KUKA KRL program: ps_b_ltb_res_c02.src, ps_b_ltb_res_c02.dat

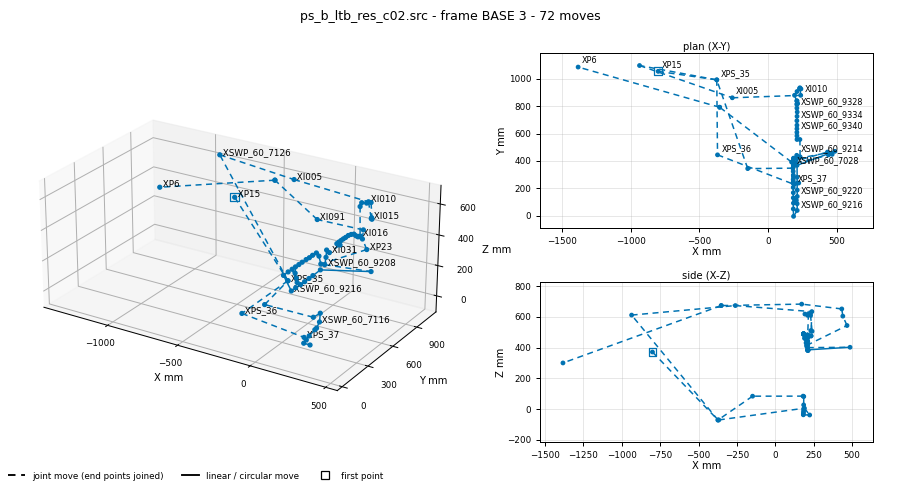
[picture p0: tool path of ps_b_ltb_res_c02.src in frame BASE 3, 72 of 73 moves have a stored position in this frame; points joined in program order, loops and branches not executed]
--- ps_b_ltb_res_c02.src ---
&ACCESS RVO1
&COMMENT Solda Axor LTB
DEF ps_b_ltb_res_c02( )

  ;FOLD INI;%{PE}%V2.2.2,%MKUKATPBASIS,%CINIT,%VCOMMON,%P
  ;FOLD BAS INI;%{PE}%V2.2.2,%MKUKATPBASIS,%CINIT,%VINIT,%P
  INTERRUPT DECL 3 WHEN $STOPMESS==TRUE DO IR_STOPM ( )
  INTERRUPT ON 3
  BAS (#INITMOV,0 )
  ;ENDFOLD
  ;FOLD A20 INI;%{E}%V2.2.2,%MKUKATPA20,%CINIT,%VINIT,%P
  IF ARC20==TRUE THEN
    A20 (ARC_INI)
    INTERRUPT DECL 6 WHEN $CYCFLAG[3]==FALSE DO A20(TECH_STOP2)
  ENDIF
  ;ENDFOLD
  ;FOLD A10 INI;%{E}%V2.2.2,%MKUKATPARC,%CINIT,%VINIT,%P
  IF A10_OPTION==#ACTIVE THEN
    INTERRUPT DECL 4 WHEN $CYCFLAG[2]==FALSE DO A10 (#APPL_ERROR)
    INTERRUPT DECL 7 WHEN A_ARC_SWI==#ACTIVE DO A10 (#ARC_SEAM)
    INTERRUPT DECL 5 WHEN A_FLY_ARC==TRUE DO A10 (#HPU_ARC)
    INTERRUPT  ON 5
    A10_INI ( )
  ENDIF
  ;ENDFOLD
  ;FOLD GRIPPER INI;%{E}%V2.2.2,%MKUKATPGRIPPER,%CINIT,%VINIT,%P
  USER_GRP(0,DUMMY,DUMMY,GDEFAULT)
  ;ENDFOLD
  ;FOLD SPOT INI;%{E}%V.2.2,%MKUKATPSPOT,%CINIT,%VINIT,%P
  USERSPOT(#INIT)
  ;ENDFOLD
  ;FOLD TOUCHSENSE INI;%{E}%V2.2.2,%MKUKATPTS,%CINIT,%VINIT,%P
  IF H70_OPTION THEN
    INTERRUPT DECL 15 WHEN $MEAS_PULSE[TOUCH_I[TOUCH_ACTIVE].IN_NR] DO H70 (6,CD0 )
    INTERRUPT DECL 16 WHEN $ZERO_MOVE DO H70 (7,CD0 )
    INTERRUPT DECL 17 WHEN $TECHPAR_C[FG_TOUCH,8]>0.5 DO H70 (8,CD0)
    H70 (1,CD0 )
  ENDIF
  ;ENDFOLD
  ;FOLD USER INI;%{P}%V2.2.2,%MKUKATPUSER,%CINIT,%VINIT,%P
  ;Make your modifications here
  ;ENDFOLD
  ;ENDFOLD

; Caracterizacao dos meios de producao
; Changes: Solda Respot - ATEGO - STB
; Versao Atual: 26/03/2016
; Ferramenta : Gun C02
; Name: P13.060-R4

chk_w3_wechs_ok ( )    ; CHECK GUN C02

IF(NOT(GHOST())) THEN
IF MaxStandMenge(3) THEN
  MaxStandmengeErreicht()
ENDIF

IF Elektrodenwechsel(3) THEN
e_Fraes3()
ENDIF
ENDIF

;FOLD OUT 868 'Perfil Livre Estacao'  State= FALSE ;%{PE}%R 4.1.16,%MKUKATPBASIS,%COUT,%VOUTX,%P 2:868, 3:'Perfil Livre Estacao', 5:FALSE, 6:
$OUT[868]=FALSE
;ENDFOLD

;FOLD PTP P15  Vel= 100 % PDAT2 Tool[1]:GUN C1 Base[3]:Atego/Axor;%{PE}%R 4.1.16,%MKUKATPBASIS,%CMOVE,%VPTP,%P 1:PTP, 2:P15, 3:, 5:100, 7:PDAT2
$BWDSTART = FALSE
PDAT_ACT=PPDAT2
BAS(#PTP_DAT)
FDAT_ACT=FP15
BAS(#FRAMES)
BAS(#VEL_PTP,100)
PTP XP15
;ENDFOLD

;FOLD ; Liga Intertravamento 1 c/ R01;%{PE}%R 4.1.16,%MKUKATPBASIS,%CCOMMENT,%VNORMAL,%P 2:Liga Intertravamento 1 c/ R01
;ENDFOLD
;FOLD ; Liga Intertravamento 10 c/ R02;%{PE}%R 4.1.16,%MKUKATPBASIS,%CCOMMENT,%VNORMAL,%P 2:Liga Intertravamento 10 c/ R02
;ENDFOLD
;FOLD Kollision.Ueberwachung_1_Ein ;%{PE}%MKUKATPUSER
COLLSTOP( 1, 1 ) ;INTERRUPTUEBERWACHT
;ENDFOLD
;FOLD Kollision.Monitoring_AREA_4_On ;%{PE}%MKUKATPUSER
COLLSTOP( 10, 1 ) ;NICHT INTERRUPTUEBERWACHT
;ENDFOLD


;FOLD ; Liga Intertravamento 3 c/ R03;%{PE}%R 4.1.16,%MKUKATPBASIS,%CCOMMENT,%VNORMAL,%P 2:Liga Intertravamento 7 c/ R03
;ENDFOLD
;FOLD Kollision.Ueberwachung_3_Ein ;%{PE}%MKUKATPUSER
COLLSTOP( 3, 1 ) ;INTERRUPTUEBERWACHT
;ENDFOLD


;FOLD PTP PS_35 CONT Vel= 100 % PDAT29 Tool[3]:GUN C02 Base[3]:Atego/Axor;%{PE}%R 4.1.16,%MKUKATPBASIS,%CMOVE,%VPTP,%P 1:PTP, 2:PS_35, 3:C_PTP, 5:100, 7:PDAT29
$BWDSTART = FALSE
PDAT_ACT=PPDAT29
BAS(#PTP_DAT)
FDAT_ACT=FPS_35
BAS(#FRAMES)
BAS(#VEL_PTP,100)
PTP XPS_35 C_PTP
;ENDFOLD
;FOLD PTP PS_36 CONT Vel= 100 % PDAT30 Tool[3]:GUN C02 Base[3]:Atego/Axor;%{PE}%R 4.1.16,%MKUKATPBASIS,%CMOVE,%VPTP,%P 1:PTP, 2:PS_36, 3:C_PTP, 5:100, 7:PDAT30
$BWDSTART = FALSE
PDAT_ACT=PPDAT30
BAS(#PTP_DAT)
FDAT_ACT=FPS_36
BAS(#FRAMES)
BAS(#VEL_PTP,100)
PTP XPS_36 C_PTP
;ENDFOLD
;FOLD PTP PS_37 CONT Vel= 100 % PDAT31 Tool[3]:GUN C02 Base[3]:Atego/Axor;%{PE}%R 4.1.16,%MKUKATPBASIS,%CMOVE,%VPTP,%P 1:PTP, 2:PS_37, 3:C_PTP, 5:100, 7:PDAT31
$BWDSTART = FALSE
PDAT_ACT=PPDAT31
BAS(#PTP_DAT)
FDAT_ACT=FPS_37
BAS(#FRAMES)
BAS(#VEL_PTP,100)
PTP XPS_37 C_PTP
;ENDFOLD
;FOLD PTP PS_38 CONT Vel= 100 % PDAT32 Tool[3]:GUN C02 Base[3]:Atego/Axor;%{PE}%R 4.1.16,%MKUKATPBASIS,%CMOVE,%VPTP,%P 1:PTP, 2:PS_38, 3:C_PTP, 5:100, 7:PDAT32
$BWDSTART = FALSE
PDAT_ACT=PPDAT32
BAS(#PTP_DAT)
FDAT_ACT=FPS_38
BAS(#FRAMES)
BAS(#VEL_PTP,100)
PTP XPS_38 C_PTP
;ENDFOLD


;FOLD LIN SWP_60_7106 CPDAT22 SPOT Gun= 3 RETR CLS PgNo1= 197 ACTIVE= 1 Tool[3]:GUN C02 Base[3]:Atego/Axor;%{PE}%R 4.1.12,%MKUKATPSPOT,%CSPOT,%VLIN,%P 1:LIN, 2:SWP_60_7106, 3:, 5:2, 7:CPDAT22, 10:3, 12:#FIRST, 14:#CLO, 16:197, 18:1, 20:0, 22:0, 24:1, 25:NORMAL
$BWDSTART = FALSE
LDAT_ACT=LCPDAT22
BAS(#CP_DAT)
FDAT_ACT=FSWP_60_7106
BAS(#FRAMES)
BAS(#VEL_CP,LCPDAT22.VEL)
S_ACT.GUN=3
S_ACT.PAIR=SDEFAULT.PAIR
S_ACT.RETR=#CLO
S_ACT.CLO_TM=1
S_ACT.PGNO1=197
S_ACT.PGNO2=SDEFAULT.PGNO2
S_ACT.PRESS1=SDEFAULT.PRESS1
S_ACT.PRESS2=SDEFAULT.PRESS2
S_READY=FALSE
LIN XSWP_60_7106
USERSPOT(#SPOT, S_ACT)
WAIT FOR S_READY
;ENDFOLD


;FOLD LIN SWP_60_7108 CPDAT23 SPOT Gun= 3 RETR CLS PgNo1= 197 ACTIVE= 1 Tool[3]:GUN C02 Base[3]:Atego/Axor;%{PE}%R 4.1.12,%MKUKATPSPOT,%CSPOT,%VLIN,%P 1:LIN, 2:SWP_60_7108, 3:, 5:2, 7:CPDAT23, 10:3, 12:#FIRST, 14:#CLO, 16:197, 18:1, 20:0, 22:0, 24:1, 25:NORMAL
$BWDSTART = FALSE
LDAT_ACT=LCPDAT23
BAS(#CP_DAT)
FDAT_ACT=FSWP_60_7108
BAS(#FRAMES)
BAS(#VEL_CP,LCPDAT23.VEL)
S_ACT.GUN=3
S_ACT.PAIR=SDEFAULT.PAIR
S_ACT.RETR=#CLO
S_ACT.CLO_TM=1
S_ACT.PGNO1=197
S_ACT.PGNO2=SDEFAULT.PGNO2
S_ACT.PRESS1=SDEFAULT.PRESS1
S_ACT.PRESS2=SDEFAULT.PRESS2
S_READY=FALSE
LIN XSWP_60_7108
USERSPOT(#SPOT, S_ACT)
WAIT FOR S_READY
;ENDFOLD

;FOLD LIN SWP_60_7110 CPDAT24 SPOT Gun= 3 RETR CLS PgNo1= 197 ACTIVE= 1 Tool[3]:GUN C02 Base[3]:Atego/Axor;%{PE}%R 4.1.12,%MKUKATPSPOT,%CSPOT,%VLIN,%P 1:LIN, 2:SWP_60_7110, 3:, 5:2, 7:CPDAT24, 10:3, 12:#FIRST, 14:#CLO, 16:197, 18:1, 20:0, 22:0, 24:1, 25:NORMAL
$BWDSTART = FALSE
LDAT_ACT=LCPDAT24
BAS(#CP_DAT)
FDAT_ACT=FSWP_60_7110
BAS(#FRAMES)
BAS(#VEL_CP,LCPDAT24.VEL)
S_ACT.GUN=3
S_ACT.PAIR=SDEFAULT.PAIR
S_ACT.RETR=#CLO
S_ACT.CLO_TM=1
S_ACT.PGNO1=197
S_ACT.PGNO2=SDEFAULT.PGNO2
S_ACT.PRESS1=SDEFAULT.PRESS1
S_ACT.PRESS2=SDEFAULT.PRESS2
S_READY=FALSE
LIN XSWP_60_7110
USERSPOT(#SPOT, S_ACT)
WAIT FOR S_READY
;ENDFOLD

;FOLD LIN SWP_60_7028 CPDAT25 SPOT Gun= 3 RETR CLS PgNo1= 197 ACTIVE= 1 Tool[3]:GUN C02 Base[3]:Atego/Axor;%{PE}%R 4.1.12,%MKUKATPSPOT,%CSPOT,%VLIN,%P 1:LIN, 2:SWP_60_7028, 3:, 5:2, 7:CPDAT25, 10:3, 12:#FIRST, 14:#CLO, 16:197, 18:1, 20:0, 22:0, 24:1, 25:NORMAL
$BWDSTART = FALSE
LDAT_ACT=LCPDAT25
BAS(#CP_DAT)
FDAT_ACT=FSWP_60_7028
BAS(#FRAMES)
BAS(#VEL_CP,LCPDAT25.VEL)
S_ACT.GUN=3
S_ACT.PAIR=SDEFAULT.PAIR
S_ACT.RETR=#CLO
S_ACT.CLO_TM=1
S_ACT.PGNO1=197
S_ACT.PGNO2=SDEFAULT.PGNO2
S_ACT.PRESS1=SDEFAULT.PRESS1
S_ACT.PRESS2=SDEFAULT.PRESS2
S_READY=FALSE
LIN XSWP_60_7028
USERSPOT(#SPOT, S_ACT)
WAIT FOR S_READY
;ENDFOLD

;FOLD LIN SWP_60_7114 CPDAT26 SPOT Gun= 3 RETR CLS PgNo1= 197 ACTIVE= 1 Tool[3]:GUN C02 Base[3]:Atego/Axor;%{PE}%R 4.1.12,%MKUKATPSPOT,%CSPOT,%VLIN,%P 1:LIN, 2:SWP_60_7114, 3:, 5:2, 7:CPDAT26, 10:3, 12:#FIRST, 14:#CLO, 16:197, 18:1, 20:0, 22:0, 24:1, 25:NORMAL
$BWDSTART = FALSE
LDAT_ACT=LCPDAT26
BAS(#CP_DAT)
FDAT_ACT=FSWP_60_7114
BAS(#FRAMES)
BAS(#VEL_CP,LCPDAT26.VEL)
S_ACT.GUN=3
S_ACT.PAIR=SDEFAULT.PAIR
S_ACT.RETR=#CLO
S_ACT.CLO_TM=1
S_ACT.PGNO1=197
S_ACT.PGNO2=SDEFAULT.PGNO2
S_ACT.PRESS1=SDEFAULT.PRESS1
S_ACT.PRESS2=SDEFAULT.PRESS2
S_READY=FALSE
LIN XSWP_60_7114
USERSPOT(#SPOT, S_ACT)
WAIT FOR S_READY
;ENDFOLD


;FOLD LIN SWP_60_7116 CPDAT27 SPOT Gun= 3 RETR CLS PgNo1= 197 ACTIVE= 1 Tool[3]:GUN C02 Base[3]:Atego/Axor;%{PE}%R 4.1.12,%MKUKATPSPOT,%CSPOT,%VLIN,%P 1:LIN, 2:SWP_60_7116, 3:, 5:2, 7:CPDAT27, 10:3, 12:#FIRST, 14:#CLO, 16:197, 18:1, 20:0, 22:0, 24:1, 25:NORMAL
$BWDSTART = FALSE
LDAT_ACT=LCPDAT27
BAS(#CP_DAT)
FDAT_ACT=FSWP_60_7116
BAS(#FRAMES)
BAS(#VEL_CP,LCPDAT27.VEL)
S_ACT.GUN=3
S_ACT.PAIR=SDEFAULT.PAIR
S_ACT.RETR=#CLO
S_ACT.CLO_TM=1
S_ACT.PGNO1=197
S_ACT.PGNO2=SDEFAULT.PGNO2
S_ACT.PRESS1=SDEFAULT.PRESS1
S_ACT.PRESS2=SDEFAULT.PRESS2
S_READY=FALSE
LIN XSWP_60_7116
USERSPOT(#SPOT, S_ACT)
WAIT FOR S_READY
;ENDFOLD


;FOLD LIN SWP_60_7120 CPDAT29 SPOT Gun= 3 RETR OPN PgNo1= 197 ACTIVE= 1 Tool[3]:GUN C02 Base[3]:Atego/Axor;%{PE}%R 4.1.12,%MKUKATPSPOT,%CSPOT,%VLIN,%P 1:LIN, 2:SWP_60_7120, 3:, 5:2, 7:CPDAT29, 10:3, 12:#FIRST, 14:#OPN, 16:197, 18:1, 20:0, 22:0, 24:1, 25:NORMAL
$BWDSTART = FALSE
LDAT_ACT=LCPDAT29
BAS(#CP_DAT)
FDAT_ACT=FSWP_60_7120
BAS(#FRAMES)
BAS(#VEL_CP,LCPDAT29.VEL)
S_ACT.GUN=3
S_ACT.PAIR=SDEFAULT.PAIR
S_ACT.RETR=#OPN
S_ACT.CLO_TM=1
S_ACT.PGNO1=197
S_ACT.PGNO2=SDEFAULT.PGNO2
S_ACT.PRESS1=SDEFAULT.PRESS1
S_ACT.PRESS2=SDEFAULT.PRESS2
S_READY=FALSE
LIN XSWP_60_7120
USERSPOT(#SPOT, S_ACT)
WAIT FOR S_READY
;ENDFOLD


;FOLD PTP SWP_60_7122  Vel= 100 % PDAT34 Tool[3]:GUN C02 Base[3]:Atego/Axor;%{PE}%R 4.1.16,%MKUKATPBASIS,%CMOVE,%VPTP,%P 1:PTP, 2:SWP_60_7122, 3:, 5:100, 7:PDAT34
$BWDSTART = FALSE
PDAT_ACT=PPDAT34
BAS(#PTP_DAT)
FDAT_ACT=FSWP_60_7122
BAS(#FRAMES)
BAS(#VEL_PTP,100)
PTP XSWP_60_7122
;ENDFOLD
;FOLD PTP SWP_60_7123  Vel= 100 % PDAT35 Tool[3]:GUN C02 Base[3]:Atego/Axor;%{PE}%R 4.1.16,%MKUKATPBASIS,%CMOVE,%VPTP,%P 1:PTP, 2:SWP_60_7123, 3:, 5:100, 7:PDAT35
$BWDSTART = FALSE
PDAT_ACT=PPDAT35
BAS(#PTP_DAT)
FDAT_ACT=FSWP_60_7123
BAS(#FRAMES)
BAS(#VEL_PTP,100)
PTP XSWP_60_7123
;ENDFOLD
;FOLD PTP SWP_60_7124  Vel= 100 % PDAT36 Tool[3]:GUN C02 Base[3]:Atego/Axor;%{PE}%R 4.1.16,%MKUKATPBASIS,%CMOVE,%VPTP,%P 1:PTP, 2:SWP_60_7124, 3:, 5:100, 7:PDAT36
$BWDSTART = FALSE
PDAT_ACT=PPDAT36
BAS(#PTP_DAT)
FDAT_ACT=FSWP_60_7124
BAS(#FRAMES)
BAS(#VEL_PTP,100)
PTP XSWP_60_7124
;ENDFOLD
;FOLD PTP SWP_60_7126  Vel= 100 % PDAT38 Tool[3]:GUN C02 Base[3]:Atego/Axor;%{PE}%R 4.1.16,%MKUKATPBASIS,%CMOVE,%VPTP,%P 1:PTP, 2:SWP_60_7126, 3:, 5:100, 7:PDAT38
$BWDSTART = FALSE
PDAT_ACT=PPDAT38
BAS(#PTP_DAT)
FDAT_ACT=FSWP_60_7126
BAS(#FRAMES)
BAS(#VEL_PTP,100)
PTP XSWP_60_7126
;ENDFOLD






;FOLD PTP l005  CONT Vel= 100 % P_OLP2 Tool[3]:Gun C02 Base[3]:Atego/Axor;%{PE}%R4.1.16,%MKUKATPBASIS,%CMOVE,%VPTP,%P 1:PTP, 2:l005, 3:C_PTP, 5:100, 7:P_OLP2
$BWDSTART = FALSE
PDAT_ACT= PP_OLP2
BAS(#PTP_DAT)
FDAT_ACT= Fl005
BAS(#FRAMES)
BAS(#VEL_PTP,100)
PTP Xl005  C_PTP
;ENDFOLD
;FOLD PTP l010  Vel= 100 % P_OLP3 Tool[3]:GUN C02 Base[3]:Atego/Axor;%{PE}%R 4.1.16,%MKUKATPBASIS,%CMOVE,%VPTP,%P 1:PTP, 2:l010, 3:, 5:100, 7:P_OLP3
$BWDSTART = FALSE
PDAT_ACT=PP_OLP3
BAS(#PTP_DAT)
FDAT_ACT=Fl010
BAS(#FRAMES)
BAS(#VEL_PTP,100)
PTP Xl010
;ENDFOLD
;FOLD PTP l015  CONT Vel= 100 % P_OLP4 Tool[3]:Gun C02 Base[3]:Atego/Axor;%{PE}%R4.1.16,%MKUKATPBASIS,%CMOVE,%VPTP,%P 1:PTP, 2:l015, 3:C_PTP, 5:100, 7:P_OLP4
$BWDSTART = FALSE
PDAT_ACT= PP_OLP4
BAS(#PTP_DAT)
FDAT_ACT= Fl015
BAS(#FRAMES)
BAS(#VEL_PTP,100)
PTP Xl015  C_PTP
;ENDFOLD

;FOLD ; SWP_60_9320;%{PE}%R 4.1.16,%MKUKATPBASIS,%CCOMMENT,%VNORMAL,%P 2:SWP_60_9320
;ENDFOLD
;FOLD LIN SWP_60_9320 L_OLP1 SPOT Gun= 3 RETR OPN PgNo1= 196 ACTIVE= 1 Tool[3]:GUN C02 Base[3]:Atego/Axor;%{PE}%R 4.1.12,%MKUKATPSPOT,%CSPOT,%VLIN,%P 1:LIN, 2:SWP_60_9320, 3:, 5:2, 7:L_OLP1, 10:3, 12:#FIRST, 14:#OPN, 16:196, 18:1, 20:0, 22:0, 24:1, 25:NORMAL
$BWDSTART = FALSE
LDAT_ACT=LL_OLP1
BAS(#CP_DAT)
FDAT_ACT=FSWP_60_9320
BAS(#FRAMES)
BAS(#VEL_CP,LL_OLP1.VEL)
S_ACT.GUN=3
S_ACT.PAIR=SDEFAULT.PAIR
S_ACT.RETR=#OPN
S_ACT.CLO_TM=1
S_ACT.PGNO1=196
S_ACT.PGNO2=SDEFAULT.PGNO2
S_ACT.PRESS1=SDEFAULT.PRESS1
S_ACT.PRESS2=SDEFAULT.PRESS2
S_READY=FALSE
LIN XSWP_60_9320
USERSPOT(#SPOT, S_ACT)
WAIT FOR S_READY
;ENDFOLD

;FOLD PTP l020  CONT Vel= 100 % P_OLP5 Tool[3]:Gun C02 Base[3]:Atego/Axor;%{PE}%R4.1.16,%MKUKATPBASIS,%CMOVE,%VPTP,%P 1:PTP, 2:l020, 3:C_PTP, 5:100, 7:P_OLP5
$BWDSTART = FALSE
PDAT_ACT= PP_OLP5
BAS(#PTP_DAT)
FDAT_ACT= Fl020
BAS(#FRAMES)
BAS(#VEL_PTP,100)
PTP Xl020  C_PTP
;ENDFOLD
;FOLD PTP l025  CONT Vel= 100 % P_OLP6 Tool[3]:Gun C02 Base[3]:Atego/Axor;%{PE}%R4.1.16,%MKUKATPBASIS,%CMOVE,%VPTP,%P 1:PTP, 2:l025, 3:C_PTP, 5:100, 7:P_OLP6
$BWDSTART = FALSE
PDAT_ACT= PP_OLP6
BAS(#PTP_DAT)
FDAT_ACT= Fl025
BAS(#FRAMES)
BAS(#VEL_PTP,100)
PTP Xl025  C_PTP
;ENDFOLD
;FOLD PTP P7 CONT Vel= 100 % PDAT7 Tool[3]:GUN C02 Base[3]:Atego/Axor;%{PE}%R 4.1.16,%MKUKATPBASIS,%CMOVE,%VPTP,%P 1:PTP, 2:P7, 3:C_PTP, 5:100, 7:PDAT7
$BWDSTART = FALSE
PDAT_ACT=PPDAT7
BAS(#PTP_DAT)
FDAT_ACT=FP7
BAS(#FRAMES)
BAS(#VEL_PTP,100)
PTP XP7 C_PTP
;ENDFOLD
;FOLD PTP l030  CONT Vel= 100 % P_OLP7 Tool[3]:Gun C02 Base[3]:Atego/Axor;%{PE}%R4.1.16,%MKUKATPBASIS,%CMOVE,%VPTP,%P 1:PTP, 2:l030, 3:C_PTP, 5:100, 7:P_OLP7
$BWDSTART = FALSE
PDAT_ACT= PP_OLP7
BAS(#PTP_DAT)
FDAT_ACT= Fl030
BAS(#FRAMES)
BAS(#VEL_PTP,100)
PTP Xl030  C_PTP
;ENDFOLD
;FOLD PTP l011  Vel= 100 % P_OLP11 Tool[3]:GUN C02 Base[3]:Atego/Axor;%{PE}%R 4.1.16,%MKUKATPBASIS,%CMOVE,%VPTP,%P 1:PTP, 2:l011, 3:, 5:100, 7:P_OLP11
$BWDSTART = FALSE
PDAT_ACT=PP_OLP11
BAS(#PTP_DAT)
FDAT_ACT=Fl011
BAS(#FRAMES)
BAS(#VEL_PTP,100)
PTP Xl011
;ENDFOLD
;FOLD PTP l016  Vel= 100 % P_OLP12 Tool[3]:GUN C02 Base[3]:Atego/Axor;%{PE}%R 4.1.16,%MKUKATPBASIS,%CMOVE,%VPTP,%P 1:PTP, 2:l016, 3:, 5:100, 7:P_OLP12
$BWDSTART = FALSE
PDAT_ACT=PP_OLP12
BAS(#PTP_DAT)
FDAT_ACT=Fl016
BAS(#FRAMES)
BAS(#VEL_PTP,100)
PTP Xl016
;ENDFOLD

;FOLD ; SWP_60_9324;%{PE}%R 4.1.16,%MKUKATPBASIS,%CCOMMENT,%VNORMAL,%P 2:SWP_60_9324
;ENDFOLD
;FOLD LIN SWP_60_9324 L_OLP2 SPOT Gun= 3 RETR CLS PgNo1= 197 ACTIVE= 1 Tool[3]:GUN C02 Base[3]:Atego/Axor;%{PE}%R 4.1.12,%MKUKATPSPOT,%CSPOT,%VLIN,%P 1:LIN, 2:SWP_60_9324, 3:, 5:2, 7:L_OLP2, 10:3, 12:#FIRST, 14:#CLO, 16:197, 18:1, 20:0, 22:0, 24:1, 25:NORMAL
$BWDSTART = FALSE
LDAT_ACT=LL_OLP2
BAS(#CP_DAT)
FDAT_ACT=FSWP_60_9324
BAS(#FRAMES)
BAS(#VEL_CP,LL_OLP2.VEL)
S_ACT.GUN=3
S_ACT.PAIR=SDEFAULT.PAIR
S_ACT.RETR=#CLO
S_ACT.CLO_TM=1
S_ACT.PGNO1=197
S_ACT.PGNO2=SDEFAULT.PGNO2
S_ACT.PRESS1=SDEFAULT.PRESS1
S_ACT.PRESS2=SDEFAULT.PRESS2
S_READY=FALSE
LIN XSWP_60_9324
USERSPOT(#SPOT, S_ACT)
WAIT FOR S_READY
;ENDFOLD

;FOLD ; SWP_60_9236;%{PE}%R 4.1.16,%MKUKATPBASIS,%CCOMMENT,%VNORMAL,%P 2:SWP_60_9236
;ENDFOLD
;FOLD LIN SWP_60_9326 L_OLP3 SPOT Gun= 3 RETR CLS PgNo1= 197 ACTIVE= 1 Tool[3]:GUN C02 Base[3]:Atego/Axor;%{PE}%R 4.1.12,%MKUKATPSPOT,%CSPOT,%VLIN,%P 1:LIN, 2:SWP_60_9326, 3:, 5:2, 7:L_OLP3, 10:3, 12:#FIRST, 14:#CLO, 16:197, 18:1, 20:0, 22:0, 24:1, 25:NORMAL1
$BWDSTART = FALSE
LDAT_ACT=LL_OLP3
BAS(#CP_DAT)
FDAT_ACT=FSWP_60_9326
BAS(#FRAMES)
BAS(#VEL_CP,LL_OLP3.VEL)
S_ACT.GUN=3
S_ACT.PAIR=SDEFAULT.PAIR
S_ACT.RETR=#CLO
S_ACT.CLO_TM=1
S_ACT.PGNO1=197
S_ACT.PGNO2=SDEFAULT.PGNO2
S_ACT.PRESS1=SDEFAULT.PRESS1
S_ACT.PRESS2=SDEFAULT.PRESS2
S_READY=FALSE
LIN XSWP_60_9326
USERSPOT(#SPOT, S_ACT)
WAIT FOR S_READY
;ENDFOLD

;FOLD ; SWP_60_9328;%{PE}%R 4.1.16,%MKUKATPBASIS,%CCOMMENT,%VNORMAL,%P 2:SWP_60_9328
;ENDFOLD
;FOLD LIN SWP_60_9328 L_OLP4 SPOT Gun= 3 RETR CLS PgNo1= 197 ACTIVE= 1 Tool[3]:GUN C02 Base[3]:Atego/Axor;%{PE}%R 4.1.12,%MKUKATPSPOT,%CSPOT,%VLIN,%P 1:LIN, 2:SWP_60_9328, 3:, 5:2, 7:L_OLP4, 10:3, 12:#FIRST, 14:#CLO, 16:197, 18:1, 20:0, 22:0, 24:1, 25:NORMAL2
$BWDSTART = FALSE
LDAT_ACT=LL_OLP4
BAS(#CP_DAT)
FDAT_ACT=FSWP_60_9328
BAS(#FRAMES)
BAS(#VEL_CP,LL_OLP4.VEL)
S_ACT.GUN=3
S_ACT.PAIR=SDEFAULT.PAIR
S_ACT.RETR=#CLO
S_ACT.CLO_TM=1
S_ACT.PGNO1=197
S_ACT.PGNO2=SDEFAULT.PGNO2
S_ACT.PRESS1=SDEFAULT.PRESS1
S_ACT.PRESS2=SDEFAULT.PRESS2
S_READY=FALSE
LIN XSWP_60_9328
USERSPOT(#SPOT, S_ACT)
WAIT FOR S_READY
;ENDFOLD

;FOLD ; SWP_60_9330;%{PE}%R 4.1.16,%MKUKATPBASIS,%CCOMMENT,%VNORMAL,%P 2:SWP_60_9330
;ENDFOLD
;FOLD LIN SWP_60_9330 L_OLP5 SPOT Gun= 3 RETR CLS PgNo1= 197 ACTIVE= 1 Tool[3]:GUN C02 Base[3]:Atego/Axor;%{PE}%R 4.1.12,%MKUKATPSPOT,%CSPOT,%VLIN,%P 1:LIN, 2:SWP_60_9330, 3:, 5:2, 7:L_OLP5, 10:3, 12:#FIRST, 14:#CLO, 16:197, 18:1, 20:0, 22:0, 24:1, 25:NORMAL3
$BWDSTART = FALSE
LDAT_ACT=LL_OLP5
BAS(#CP_DAT)
FDAT_ACT=FSWP_60_9330
BAS(#FRAMES)
BAS(#VEL_CP,LL_OLP5.VEL)
S_ACT.GUN=3
S_ACT.PAIR=SDEFAULT.PAIR
S_ACT.RETR=#CLO
S_ACT.CLO_TM=1
S_ACT.PGNO1=197
S_ACT.PGNO2=SDEFAULT.PGNO2
S_ACT.PRESS1=SDEFAULT.PRESS1
S_ACT.PRESS2=SDEFAULT.PRESS2
S_READY=FALSE
LIN XSWP_60_9330
USERSPOT(#SPOT, S_ACT)
WAIT FOR S_READY
;ENDFOLD

;FOLD ; SWP_60_9332;%{PE}%R 4.1.16,%MKUKATPBASIS,%CCOMMENT,%VNORMAL,%P 2:SWP_60_9332
;ENDFOLD
;FOLD LIN SWP_60_9332 L_OLP6 SPOT Gun= 3 RETR CLS PgNo1= 197 ACTIVE= 1 Tool[3]:GUN C02 Base[3]:Atego/Axor;%{PE}%R 4.1.12,%MKUKATPSPOT,%CSPOT,%VLIN,%P 1:LIN, 2:SWP_60_9332, 3:, 5:2, 7:L_OLP6, 10:3, 12:#FIRST, 14:#CLO, 16:197, 18:1, 20:0, 22:0, 24:1, 25:NORMAL4
$BWDSTART = FALSE
LDAT_ACT=LL_OLP6
BAS(#CP_DAT)
FDAT_ACT=FSWP_60_9332
BAS(#FRAMES)
BAS(#VEL_CP,LL_OLP6.VEL)
S_ACT.GUN=3
S_ACT.PAIR=SDEFAULT.PAIR
S_ACT.RETR=#CLO
S_ACT.CLO_TM=1
S_ACT.PGNO1=197
S_ACT.PGNO2=SDEFAULT.PGNO2
S_ACT.PRESS1=SDEFAULT.PRESS1
S_ACT.PRESS2=SDEFAULT.PRESS2
S_READY=FALSE
LIN XSWP_60_9332
USERSPOT(#SPOT, S_ACT)
WAIT FOR S_READY
;ENDFOLD

;FOLD ; SWP_60_9334;%{PE}%R 4.1.16,%MKUKATPBASIS,%CCOMMENT,%VNORMAL,%P 2:SWP_60_9334
;ENDFOLD
;FOLD LIN SWP_60_9334 L_OLP7 SPOT Gun= 3 RETR CLS PgNo1= 197 ACTIVE= 1 Tool[3]:GUN C02 Base[3]:Atego/Axor;%{PE}%R 4.1.12,%MKUKATPSPOT,%CSPOT,%VLIN,%P 1:LIN, 2:SWP_60_9334, 3:, 5:2, 7:L_OLP7, 10:3, 12:#FIRST, 14:#CLO, 16:197, 18:1, 20:0, 22:0, 24:1, 25:NORMAL5
$BWDSTART = FALSE
LDAT_ACT=LL_OLP7
BAS(#CP_DAT)
FDAT_ACT=FSWP_60_9334
BAS(#FRAMES)
BAS(#VEL_CP,LL_OLP7.VEL)
S_ACT.GUN=3
S_ACT.PAIR=SDEFAULT.PAIR
S_ACT.RETR=#CLO
S_ACT.CLO_TM=1
S_ACT.PGNO1=197
S_ACT.PGNO2=SDEFAULT.PGNO2
S_ACT.PRESS1=SDEFAULT.PRESS1
S_ACT.PRESS2=SDEFAULT.PRESS2
S_READY=FALSE
LIN XSWP_60_9334
USERSPOT(#SPOT, S_ACT)
WAIT FOR S_READY
;ENDFOLD

;FOLD ; SWP_60_9336;%{PE}%R 4.1.16,%MKUKATPBASIS,%CCOMMENT,%VNORMAL,%P 2:SWP_60_9336
;ENDFOLD
;FOLD LIN SWP_60_9336 L_OLP8 SPOT Gun= 3 RETR CLS PgNo1= 197 ACTIVE= 1 Tool[3]:GUN C02 Base[3]:Atego/Axor;%{PE}%R 4.1.12,%MKUKATPSPOT,%CSPOT,%VLIN,%P 1:LIN, 2:SWP_60_9336, 3:, 5:2, 7:L_OLP8, 10:3, 12:#FIRST, 14:#CLO, 16:197, 18:1, 20:0, 22:0, 24:1, 25:NORMAL6
$BWDSTART = FALSE
LDAT_ACT=LL_OLP8
BAS(#CP_DAT)
FDAT_ACT=FSWP_60_9336
BAS(#FRAMES)
BAS(#VEL_CP,LL_OLP8.VEL)
S_ACT.GUN=3
S_ACT.PAIR=SDEFAULT.PAIR
S_ACT.RETR=#CLO
S_ACT.CLO_TM=1
S_ACT.PGNO1=197
S_ACT.PGNO2=SDEFAULT.PGNO2
S_ACT.PRESS1=SDEFAULT.PRESS1
S_ACT.PRESS2=SDEFAULT.PRESS2
S_READY=FALSE
LIN XSWP_60_9336
USERSPOT(#SPOT, S_ACT)
WAIT FOR S_READY
;ENDFOLD

;FOLD ; SWP_60_9338;%{PE}%R 4.1.16,%MKUKATPBASIS,%CCOMMENT,%VNORMAL,%P 2:SWP_60_9338
;ENDFOLD
;FOLD LIN SWP_60_9338 L_OLP9 SPOT Gun= 3 RETR CLS PgNo1= 197 ACTIVE= 1 Tool[3]:GUN C02 Base[3]:Atego/Axor;%{PE}%R 4.1.12,%MKUKATPSPOT,%CSPOT,%VLIN,%P 1:LIN, 2:SWP_60_9338, 3:, 5:2, 7:L_OLP9, 10:3, 12:#FIRST, 14:#CLO, 16:197, 18:1, 20:0, 22:0, 24:1, 25:NORMAL7
$BWDSTART = FALSE
LDAT_ACT=LL_OLP9
BAS(#CP_DAT)
FDAT_ACT=FSWP_60_9338
BAS(#FRAMES)
BAS(#VEL_CP,LL_OLP9.VEL)
S_ACT.GUN=3
S_ACT.PAIR=SDEFAULT.PAIR
S_ACT.RETR=#CLO
S_ACT.CLO_TM=1
S_ACT.PGNO1=197
S_ACT.PGNO2=SDEFAULT.PGNO2
S_ACT.PRESS1=SDEFAULT.PRESS1
S_ACT.PRESS2=SDEFAULT.PRESS2
S_READY=FALSE
LIN XSWP_60_9338
USERSPOT(#SPOT, S_ACT)
WAIT FOR S_READY
;ENDFOLD

;FOLD ; SWP_60_9340;%{PE}%R 4.1.16,%MKUKATPBASIS,%CCOMMENT,%VNORMAL,%P 2:SWP_60_9340
;ENDFOLD
;FOLD LIN SWP_60_9340 L_OLP10 SPOT Gun= 3 RETR CLS PgNo1= 197 ACTIVE= 1 Tool[3]:GUN C02 Base[3]:Atego/Axor;%{PE}%R 4.1.12,%MKUKATPSPOT,%CSPOT,%VLIN,%P 1:LIN, 2:SWP_60_9340, 3:, 5:2, 7:L_OLP10, 10:3, 12:#FIRST, 14:#CLO, 16:197, 18:1, 20:0, 22:0, 24:1, 25:NORMAL8
$BWDSTART = FALSE
LDAT_ACT=LL_OLP10
BAS(#CP_DAT)
FDAT_ACT=FSWP_60_9340
BAS(#FRAMES)
BAS(#VEL_CP,LL_OLP10.VEL)
S_ACT.GUN=3
S_ACT.PAIR=SDEFAULT.PAIR
S_ACT.RETR=#CLO
S_ACT.CLO_TM=1
S_ACT.PGNO1=197
S_ACT.PGNO2=SDEFAULT.PGNO2
S_ACT.PRESS1=SDEFAULT.PRESS1
S_ACT.PRESS2=SDEFAULT.PRESS2
S_READY=FALSE
LIN XSWP_60_9340
USERSPOT(#SPOT, S_ACT)
WAIT FOR S_READY
;ENDFOLD

;FOLD ; SWP_60_9342;%{PE}%R 4.1.16,%MKUKATPBASIS,%CCOMMENT,%VNORMAL,%P 2:SWP_60_9342
;ENDFOLD
;FOLD LIN SWP_60_9342 L_OLP11 SPOT Gun= 3 RETR CLS PgNo1= 197 ACTIVE= 1 Tool[3]:GUN C02 Base[3]:Atego/Axor;%{PE}%R 4.1.12,%MKUKATPSPOT,%CSPOT,%VLIN,%P 1:LIN, 2:SWP_60_9342, 3:, 5:2, 7:L_OLP11, 10:3, 12:#FIRST, 14:#CLO, 16:197, 18:1, 20:0, 22:0, 24:1, 25:NORMAL9
$BWDSTART = FALSE
LDAT_ACT=LL_OLP11
BAS(#CP_DAT)
FDAT_ACT=FSWP_60_9342
BAS(#FRAMES)
BAS(#VEL_CP,LL_OLP11.VEL)
S_ACT.GUN=3
S_ACT.PAIR=SDEFAULT.PAIR
S_ACT.RETR=#CLO
S_ACT.CLO_TM=1
S_ACT.PGNO1=197
S_ACT.PGNO2=SDEFAULT.PGNO2
S_ACT.PRESS1=SDEFAULT.PRESS1
S_ACT.PRESS2=SDEFAULT.PRESS2
S_READY=FALSE
LIN XSWP_60_9342
USERSPOT(#SPOT, S_ACT)
WAIT FOR S_READY
;ENDFOLD

;FOLD ; SWP_60_9344;%{PE}%R 4.1.16,%MKUKATPBASIS,%CCOMMENT,%VNORMAL,%P 2:SWP_60_9344
;ENDFOLD
;FOLD LIN SWP_60_9344 L_OLP12 SPOT Gun= 3 RETR OPN PgNo1= 197 ACTIVE= 1 Tool[3]:GUN C02 Base[3]:Atego/Axor;%{PE}%R 4.1.12,%MKUKATPSPOT,%CSPOT,%VLIN,%P 1:LIN, 2:SWP_60_9344, 3:, 5:2, 7:L_OLP12, 10:3, 12:#FIRST, 14:#OPN, 16:197, 18:1, 20:0, 22:0, 24:1, 25:NORMAL10
$BWDSTART = FALSE
LDAT_ACT=LL_OLP12
BAS(#CP_DAT)
FDAT_ACT=FSWP_60_9344
BAS(#FRAMES)
BAS(#VEL_CP,LL_OLP12.VEL)
S_ACT.GUN=3
S_ACT.PAIR=SDEFAULT.PAIR
S_ACT.RETR=#OPN
S_ACT.CLO_TM=1
S_ACT.PGNO1=197
S_ACT.PGNO2=SDEFAULT.PGNO2
S_ACT.PRESS1=SDEFAULT.PRESS1
S_ACT.PRESS2=SDEFAULT.PRESS2
S_READY=FALSE
LIN XSWP_60_9344
USERSPOT(#SPOT, S_ACT)
WAIT FOR S_READY
;ENDFOLD


;FOLD ; Liga Intertravamento 7 c/ R03 Pinca C02;%{PE}%R 4.1.16,%MKUKATPBASIS,%CCOMMENT,%VNORMAL,%P 2:Liga Intertravamento 7 c/ R03 Pinca C02
;ENDFOLD
;FOLD Kollision.Monitoring_AREA_1_On ;%{PE}%MKUKATPUSER
COLLSTOP( 7, 1 ) ;NICHT INTERRUPTUEBERWACHT
;ENDFOLD








;FOLD PTP l026 CONT Vel= 100 % P_OLP14 Tool[3] Base[3]:Atego/Axor;%{PE}%R 4.1.16,%MKUKATPBASIS,%CMOVE,%VPTP,%P 1:PTP, 2:l026, 3:C_PTP, 5:100, 7:P_OLP14
$BWDSTART = FALSE
PDAT_ACT=PP_OLP14
BAS(#PTP_DAT)
FDAT_ACT=Fl026
BAS(#FRAMES)
BAS(#VEL_PTP,100)
PTP Xl026 C_PTP
;ENDFOLD
;FOLD PTP l031 CONT Vel= 100 % P_OLP15 Tool[3] Base[3]:Atego/Axor;%{PE}%R 4.1.16,%MKUKATPBASIS,%CMOVE,%VPTP,%P 1:PTP, 2:l031, 3:C_PTP, 5:100, 7:P_OLP15
$BWDSTART = FALSE
PDAT_ACT=PP_OLP15
BAS(#PTP_DAT)
FDAT_ACT=Fl031
BAS(#FRAMES)
BAS(#VEL_PTP,100)
PTP Xl031 C_PTP
;ENDFOLD

;FOLD ; SWP_60_9214;%{PE}%R 4.1.16,%MKUKATPBASIS,%CCOMMENT,%VNORMAL,%P 2:SWP_60_9214
;ENDFOLD
;FOLD LIN SWP_60_9214 L_OLP13 SPOT Gun= 3 RETR CLS PgNo1= 197 ACTIVE= 1 Tool[3]:GUN C02 Base[3]:Atego/Axor;%{PE}%R 4.1.12,%MKUKATPSPOT,%CSPOT,%VLIN,%P 1:LIN, 2:SWP_60_9214, 3:, 5:2, 7:L_OLP13, 10:3, 12:#FIRST, 14:#CLO, 16:197, 18:1, 20:0, 22:0, 24:1, 25:NORMAL11
$BWDSTART = FALSE
LDAT_ACT=LL_OLP13
BAS(#CP_DAT)
FDAT_ACT=FSWP_60_9214
BAS(#FRAMES)
BAS(#VEL_CP,LL_OLP13.VEL)
S_ACT.GUN=3
S_ACT.PAIR=SDEFAULT.PAIR
S_ACT.RETR=#CLO
S_ACT.CLO_TM=1
S_ACT.PGNO1=197
S_ACT.PGNO2=SDEFAULT.PGNO2
S_ACT.PRESS1=SDEFAULT.PRESS1
S_ACT.PRESS2=SDEFAULT.PRESS2
S_READY=FALSE
LIN XSWP_60_9214
USERSPOT(#SPOT, S_ACT)
WAIT FOR S_READY
;ENDFOLD

;FOLD ; SWP_60_9210;%{PE}%R 4.1.16,%MKUKATPBASIS,%CCOMMENT,%VNORMAL,%P 2:SWP_60_9210
;ENDFOLD
;FOLD LIN SWP_60_9210 L_OLP14 SPOT Gun= 3 RETR CLS PgNo1= 197 ACTIVE= 1 Tool[3]:GUN C02 Base[3]:Atego/Axor;%{PE}%R 4.1.12,%MKUKATPSPOT,%CSPOT,%VLIN,%P 1:LIN, 2:SWP_60_9210, 3:, 5:2, 7:L_OLP14, 10:3, 12:#FIRST, 14:#CLO, 16:197, 18:1, 20:0, 22:0, 24:1, 25:NORMAL12
$BWDSTART = FALSE
LDAT_ACT=LL_OLP14
BAS(#CP_DAT)
FDAT_ACT=FSWP_60_9210
BAS(#FRAMES)
BAS(#VEL_CP,LL_OLP14.VEL)
S_ACT.GUN=3
S_ACT.PAIR=SDEFAULT.PAIR
S_ACT.RETR=#CLO
S_ACT.CLO_TM=1
S_ACT.PGNO1=197
S_ACT.PGNO2=SDEFAULT.PGNO2
S_ACT.PRESS1=SDEFAULT.PRESS1
S_ACT.PRESS2=SDEFAULT.PRESS2
S_READY=FALSE
LIN XSWP_60_9210
USERSPOT(#SPOT, S_ACT)
WAIT FOR S_READY
;ENDFOLD

;FOLD ; SWP_60_9208;%{PE}%R 4.1.16,%MKUKATPBASIS,%CCOMMENT,%VNORMAL,%P 2:SWP_60_9208
;ENDFOLD
;FOLD LIN SWP_60_9208 L_OLP15 SPOT Gun= 3 RETR CLS PgNo1= 197 ACTIVE= 1 Tool[3]:GUN C02 Base[3]:Atego/Axor;%{PE}%R 4.1.12,%MKUKATPSPOT,%CSPOT,%VLIN,%P 1:LIN, 2:SWP_60_9208, 3:, 5:2, 7:L_OLP15, 10:3, 12:#FIRST, 14:#CLO, 16:197, 18:1, 20:0, 22:0, 24:1, 25:NORMAL13
$BWDSTART = FALSE
LDAT_ACT=LL_OLP15
BAS(#CP_DAT)
FDAT_ACT=FSWP_60_9208
BAS(#FRAMES)
BAS(#VEL_CP,LL_OLP15.VEL)
S_ACT.GUN=3
S_ACT.PAIR=SDEFAULT.PAIR
S_ACT.RETR=#CLO
S_ACT.CLO_TM=1
S_ACT.PGNO1=197
S_ACT.PGNO2=SDEFAULT.PGNO2
S_ACT.PRESS1=SDEFAULT.PRESS1
S_ACT.PRESS2=SDEFAULT.PRESS2
S_READY=FALSE
LIN XSWP_60_9208
USERSPOT(#SPOT, S_ACT)
WAIT FOR S_READY
;ENDFOLD



;FOLD PTP P17  Vel= 100 % PDAT5 Tool[1]:GUN C1 Base[3]:Atego/Axor;%{PE}%R 4.1.16,%MKUKATPBASIS,%CMOVE,%VPTP,%P 1:PTP, 2:P17, 3:, 5:100, 7:PDAT5
$BWDSTART = FALSE
PDAT_ACT=PPDAT5
BAS(#PTP_DAT)
FDAT_ACT=FP17
BAS(#FRAMES)
BAS(#VEL_PTP,100)
PTP XP17
;ENDFOLD

;FOLD ; SWP_60_9230;%{PE}%R 4.1.16,%MKUKATPBASIS,%CCOMMENT,%VNORMAL,%P 2:SWP_60_9230
;ENDFOLD
;FOLD LIN SWP_60_9230 L_OLP16 SPOT Gun= 3 RETR CLS PgNo1= 199 ACTIVE= 1 Tool[3]:GUN C02 Base[3]:Atego/Axor;%{PE}%R 4.1.12,%MKUKATPSPOT,%CSPOT,%VLIN,%P 1:LIN, 2:SWP_60_9230, 3:, 5:2, 7:L_OLP16, 10:3, 12:#FIRST, 14:#CLO, 16:199, 18:1, 20:0, 22:0, 24:1, 25:NORMAL13
$BWDSTART = FALSE
LDAT_ACT=LL_OLP16
BAS(#CP_DAT)
FDAT_ACT=FSWP_60_9230
BAS(#FRAMES)
BAS(#VEL_CP,LL_OLP16.VEL)
S_ACT.GUN=3
S_ACT.PAIR=SDEFAULT.PAIR
S_ACT.RETR=#CLO
S_ACT.CLO_TM=1
S_ACT.PGNO1=199
S_ACT.PGNO2=SDEFAULT.PGNO2
S_ACT.PRESS1=SDEFAULT.PRESS1
S_ACT.PRESS2=SDEFAULT.PRESS2
S_READY=FALSE
LIN XSWP_60_9230
USERSPOT(#SPOT, S_ACT)
WAIT FOR S_READY
;ENDFOLD

;FOLD ; SWP_60_9232;%{PE}%R 4.1.16,%MKUKATPBASIS,%CCOMMENT,%VNORMAL,%P 2:SWP_60_9232
;ENDFOLD
;FOLD LIN SWP_60_9232 L_OLP17 SPOT Gun= 3 RETR CLS PgNo1= 199 ACTIVE= 1 Tool[3]:GUN C02 Base[3]:Atego/Axor;%{PE}%R 4.1.12,%MKUKATPSPOT,%CSPOT,%VLIN,%P 1:LIN, 2:SWP_60_9232, 3:, 5:2, 7:L_OLP17, 10:3, 12:#FIRST, 14:#CLO, 16:199, 18:1, 20:0, 22:0, 24:1, 25:NORMAL14
$BWDSTART = FALSE
LDAT_ACT=LL_OLP17
BAS(#CP_DAT)
FDAT_ACT=FSWP_60_9232
BAS(#FRAMES)
BAS(#VEL_CP,LL_OLP17.VEL)
S_ACT.GUN=3
S_ACT.PAIR=SDEFAULT.PAIR
S_ACT.RETR=#CLO
S_ACT.CLO_TM=1
S_ACT.PGNO1=199
S_ACT.PGNO2=SDEFAULT.PGNO2
S_ACT.PRESS1=SDEFAULT.PRESS1
S_ACT.PRESS2=SDEFAULT.PRESS2
S_READY=FALSE
LIN XSWP_60_9232
USERSPOT(#SPOT, S_ACT)
WAIT FOR S_READY
;ENDFOLD

;FOLD ; SWP_60_9224;%{PE}%R 4.1.16,%MKUKATPBASIS,%CCOMMENT,%VNORMAL,%P 2:SWP_60_9224
;ENDFOLD
;FOLD LIN SWP_60_9224 L_OLP18 SPOT Gun= 3 RETR CLS PgNo1= 199 ACTIVE= 1 Tool[3]:GUN C02 Base[3]:Atego/Axor;%{PE}%R 4.1.12,%MKUKATPSPOT,%CSPOT,%VLIN,%P 1:LIN, 2:SWP_60_9224, 3:, 5:2, 7:L_OLP18, 10:3, 12:#FIRST, 14:#CLO, 16:199, 18:1, 20:0, 22:0, 24:1, 25:NORMAL14
$BWDSTART = FALSE
LDAT_ACT=LL_OLP18
BAS(#CP_DAT)
FDAT_ACT=FSWP_60_9224
BAS(#FRAMES)
BAS(#VEL_CP,LL_OLP18.VEL)
S_ACT.GUN=3
S_ACT.PAIR=SDEFAULT.PAIR
S_ACT.RETR=#CLO
S_ACT.CLO_TM=1
S_ACT.PGNO1=199
S_ACT.PGNO2=SDEFAULT.PGNO2
S_ACT.PRESS1=SDEFAULT.PRESS1
S_ACT.PRESS2=SDEFAULT.PRESS2
S_READY=FALSE
LIN XSWP_60_9224
USERSPOT(#SPOT, S_ACT)
WAIT FOR S_READY
;ENDFOLD

;FOLD ; SWP_60_9222;%{PE}%R 4.1.16,%MKUKATPBASIS,%CCOMMENT,%VNORMAL,%P 2:SWP_60_9222
;ENDFOLD
;FOLD LIN SWP_60_9222 L_OLP19 SPOT Gun= 3 RETR CLS PgNo1= 199 ACTIVE= 1 Tool[3]:GUN C02 Base[3]:Atego/Axor;%{PE}%R 4.1.12,%MKUKATPSPOT,%CSPOT,%VLIN,%P 1:LIN, 2:SWP_60_9222, 3:, 5:2, 7:L_OLP19, 10:3, 12:#FIRST, 14:#CLO, 16:199, 18:1, 20:0, 22:0, 24:1, 25:NORMAL14
$BWDSTART = FALSE
LDAT_ACT=LL_OLP19
BAS(#CP_DAT)
FDAT_ACT=FSWP_60_9222
BAS(#FRAMES)
BAS(#VEL_CP,LL_OLP19.VEL)
S_ACT.GUN=3
S_ACT.PAIR=SDEFAULT.PAIR
S_ACT.RETR=#CLO
S_ACT.CLO_TM=1
S_ACT.PGNO1=199
S_ACT.PGNO2=SDEFAULT.PGNO2
S_ACT.PRESS1=SDEFAULT.PRESS1
S_ACT.PRESS2=SDEFAULT.PRESS2
S_READY=FALSE
LIN XSWP_60_9222
USERSPOT(#SPOT, S_ACT)
WAIT FOR S_READY
;ENDFOLD

;FOLD ; SWP_60_9220;%{PE}%R 4.1.16,%MKUKATPBASIS,%CCOMMENT,%VNORMAL,%P 2:SWP_60_9220
;ENDFOLD
;FOLD LIN SWP_60_9220 L_OLP20 SPOT Gun= 3 RETR CLS PgNo1= 199 ACTIVE= 1 Tool[3]:GUN C02 Base[3]:Atego/Axor;%{PE}%R 4.1.12,%MKUKATPSPOT,%CSPOT,%VLIN,%P 1:LIN, 2:SWP_60_9220, 3:, 5:2, 7:L_OLP20, 10:3, 12:#FIRST, 14:#CLO, 16:199, 18:1, 20:0, 22:0, 24:1, 25:NORMAL14
$BWDSTART = FALSE
LDAT_ACT=LL_OLP20
BAS(#CP_DAT)
FDAT_ACT=FSWP_60_9220
BAS(#FRAMES)
BAS(#VEL_CP,LL_OLP20.VEL)
S_ACT.GUN=3
S_ACT.PAIR=SDEFAULT.PAIR
S_ACT.RETR=#CLO
S_ACT.CLO_TM=1
S_ACT.PGNO1=199
S_ACT.PGNO2=SDEFAULT.PGNO2
S_ACT.PRESS1=SDEFAULT.PRESS1
S_ACT.PRESS2=SDEFAULT.PRESS2
S_READY=FALSE
LIN XSWP_60_9220
USERSPOT(#SPOT, S_ACT)
WAIT FOR S_READY
;ENDFOLD





;FOLD ; SWP_60_9218;%{PE}%R 4.1.16,%MKUKATPBASIS,%CCOMMENT,%VNORMAL,%P 2:SWP_60_9218
;ENDFOLD
;FOLD LIN SWP_60_9218 CPDAT8 SPOT Gun= 3 RETR CLS PgNo1= 197 ACTIVE= 1 Tool[3]:GUN C02 Base[3]:Atego/Axor;%{PE}%R 4.1.12,%MKUKATPSPOT,%CSPOT,%VLIN,%P 1:LIN, 2:SWP_60_9218, 3:, 5:2, 7:CPDAT8, 10:3, 12:#FIRST, 14:#CLO, 16:197, 18:1, 20:0, 22:0, 24:1, 25:NORMAL1
$BWDSTART = FALSE
LDAT_ACT=LCPDAT8
BAS(#CP_DAT)
FDAT_ACT=FSWP_60_9218
BAS(#FRAMES)
BAS(#VEL_CP,LCPDAT8.VEL)
S_ACT.GUN=3
S_ACT.PAIR=SDEFAULT.PAIR
S_ACT.RETR=#CLO
S_ACT.CLO_TM=1
S_ACT.PGNO1=197
S_ACT.PGNO2=SDEFAULT.PGNO2
S_ACT.PRESS1=SDEFAULT.PRESS1
S_ACT.PRESS2=SDEFAULT.PRESS2
S_READY=FALSE
LIN XSWP_60_9218
USERSPOT(#SPOT, S_ACT)
WAIT FOR S_READY
;ENDFOLD

;FOLD ; SWP_60_9216;%{PE}%R 4.1.16,%MKUKATPBASIS,%CCOMMENT,%VNORMAL,%P 2:SWP_60_9216
;ENDFOLD
;FOLD LIN SWP_60_9216 CPDAT10 SPOT Gun= 3 RETR CLS PgNo1= 197 ACTIVE= 1 Tool[3]:GUN C02 Base[3]:Atego/Axor;%{PE}%R 4.1.12,%MKUKATPSPOT,%CSPOT,%VLIN,%P 1:LIN, 2:SWP_60_9216, 3:, 5:2, 7:CPDAT10, 10:3, 12:#FIRST, 14:#CLO, 16:197, 18:1, 20:0, 22:0, 24:1, 25:NORMAL1
$BWDSTART = FALSE
LDAT_ACT=LCPDAT10
BAS(#CP_DAT)
FDAT_ACT=FSWP_60_9216
BAS(#FRAMES)
BAS(#VEL_CP,LCPDAT10.VEL)
S_ACT.GUN=3
S_ACT.PAIR=SDEFAULT.PAIR
S_ACT.RETR=#CLO
S_ACT.CLO_TM=1
S_ACT.PGNO1=197
S_ACT.PGNO2=SDEFAULT.PGNO2
S_ACT.PRESS1=SDEFAULT.PRESS1
S_ACT.PRESS2=SDEFAULT.PRESS2
S_READY=FALSE
LIN XSWP_60_9216
USERSPOT(#SPOT, S_ACT)
WAIT FOR S_READY
;ENDFOLD


;FOLD ; SWP_60_9257;%{PE}%R 4.1.16,%MKUKATPBASIS,%CCOMMENT,%VNORMAL,%P 2:SWP_60_9257
;ENDFOLD
;FOLD LIN SWP_60_9257 L_OLP36 SPOT Gun= 3 RETR CLS PgNo1= 197 ACTIVE= 1 Tool[3]:GUN C02 Base[3]:Atego/Axor;%{PE}%R 4.1.12,%MKUKATPSPOT,%CSPOT,%VLIN,%P 1:LIN, 2:SWP_60_9257, 3:, 5:2, 7:L_OLP36, 10:3, 12:#FIRST, 14:#CLO, 16:197, 18:1, 20:0, 22:0, 24:1, 25:NORMAL34
$BWDSTART = FALSE
LDAT_ACT=LL_OLP36
BAS(#CP_DAT)
FDAT_ACT=FSWP_60_9257
BAS(#FRAMES)
BAS(#VEL_CP,LL_OLP36.VEL)
S_ACT.GUN=3
S_ACT.PAIR=SDEFAULT.PAIR
S_ACT.RETR=#CLO
S_ACT.CLO_TM=1
S_ACT.PGNO1=197
S_ACT.PGNO2=SDEFAULT.PGNO2
S_ACT.PRESS1=SDEFAULT.PRESS1
S_ACT.PRESS2=SDEFAULT.PRESS2
S_READY=FALSE
LIN XSWP_60_9257
USERSPOT(#SPOT, S_ACT)
WAIT FOR S_READY
;ENDFOLD

;FOLD ; SWP_60_9256;%{PE}%R 4.1.16,%MKUKATPBASIS,%CCOMMENT,%VNORMAL,%P 2:SWP_60_9256
;ENDFOLD
;FOLD LIN SWP_60_9256 L_OLP37 SPOT Gun= 3 RETR CLS PgNo1= 197 ACTIVE= 1 Tool[3]:GUN C02 Base[3]:Atego/Axor;%{PE}%R 4.1.12,%MKUKATPSPOT,%CSPOT,%VLIN,%P 1:LIN, 2:SWP_60_9256, 3:, 5:2, 7:L_OLP37, 10:3, 12:#FIRST, 14:#CLO, 16:197, 18:1, 20:0, 22:0, 24:1, 25:NORMAL35
$BWDSTART = FALSE
LDAT_ACT=LL_OLP37
BAS(#CP_DAT)
FDAT_ACT=FSWP_60_9256
BAS(#FRAMES)
BAS(#VEL_CP,LL_OLP37.VEL)
S_ACT.GUN=3
S_ACT.PAIR=SDEFAULT.PAIR
S_ACT.RETR=#CLO
S_ACT.CLO_TM=1
S_ACT.PGNO1=197
S_ACT.PGNO2=SDEFAULT.PGNO2
S_ACT.PRESS1=SDEFAULT.PRESS1
S_ACT.PRESS2=SDEFAULT.PRESS2
S_READY=FALSE
LIN XSWP_60_9256
USERSPOT(#SPOT, S_ACT)
WAIT FOR S_READY
;ENDFOLD

;FOLD ; SWP_60_9254;%{PE}%R 4.1.16,%MKUKATPBASIS,%CCOMMENT,%VNORMAL,%P 2:SWP_60_9254
;ENDFOLD
;FOLD LIN SWP_60_9254 L_OLP38 SPOT Gun= 3 RETR CLS PgNo1= 197 ACTIVE= 1 Tool[3]:GUN C02 Base[3]:Atego/Axor;%{PE}%R 4.1.12,%MKUKATPSPOT,%CSPOT,%VLIN,%P 1:LIN, 2:SWP_60_9254, 3:, 5:2, 7:L_OLP38, 10:3, 12:#FIRST, 14:#CLO, 16:197, 18:1, 20:0, 22:0, 24:1, 25:NORMAL36
$BWDSTART = FALSE
LDAT_ACT=LL_OLP38
BAS(#CP_DAT)
FDAT_ACT=FSWP_60_9254
BAS(#FRAMES)
BAS(#VEL_CP,LL_OLP38.VEL)
S_ACT.GUN=3
S_ACT.PAIR=SDEFAULT.PAIR
S_ACT.RETR=#CLO
S_ACT.CLO_TM=1
S_ACT.PGNO1=197
S_ACT.PGNO2=SDEFAULT.PGNO2
S_ACT.PRESS1=SDEFAULT.PRESS1
S_ACT.PRESS2=SDEFAULT.PRESS2
S_READY=FALSE
LIN XSWP_60_9254
USERSPOT(#SPOT, S_ACT)
WAIT FOR S_READY
;ENDFOLD




;FOLD ; SWP_60_9308;%{PE}%R 4.1.16,%MKUKATPBASIS,%CCOMMENT,%VNORMAL,%P 2:SWP_60_9308
;ENDFOLD
;FOLD LIN SWP_60_9308 L_OLP39 SPOT Gun= 3 RETR CLS PgNo1= 199 ACTIVE= 1 Tool[3]:GUN C02 Base[3]:Atego/Axor;%{PE}%R 4.1.12,%MKUKATPSPOT,%CSPOT,%VLIN,%P 1:LIN, 2:SWP_60_9308, 3:, 5:2, 7:L_OLP39, 10:3, 12:#FIRST, 14:#CLO, 16:199, 18:1, 20:0, 22:0, 24:1, 25:NORMAL36
$BWDSTART = FALSE
LDAT_ACT=LL_OLP39
BAS(#CP_DAT)
FDAT_ACT=FSWP_60_9308
BAS(#FRAMES)
BAS(#VEL_CP,LL_OLP39.VEL)
S_ACT.GUN=3
S_ACT.PAIR=SDEFAULT.PAIR
S_ACT.RETR=#CLO
S_ACT.CLO_TM=1
S_ACT.PGNO1=199
S_ACT.PGNO2=SDEFAULT.PGNO2
S_ACT.PRESS1=SDEFAULT.PRESS1
S_ACT.PRESS2=SDEFAULT.PRESS2
S_READY=FALSE
LIN XSWP_60_9308
USERSPOT(#SPOT, S_ACT)
WAIT FOR S_READY
;ENDFOLD

;FOLD ; SWP_60_9310;%{PE}%R 4.1.16,%MKUKATPBASIS,%CCOMMENT,%VNORMAL,%P 2:SWP_60_9310
;ENDFOLD
;FOLD LIN SWP_60_9310 L_OLP40 SPOT Gun= 3 RETR CLS PgNo1= 199 ACTIVE= 1 Tool[3]:GUN C02 Base[3]:Atego/Axor;%{PE}%R 4.1.12,%MKUKATPSPOT,%CSPOT,%VLIN,%P 1:LIN, 2:SWP_60_9310, 3:, 5:2, 7:L_OLP40, 10:3, 12:#FIRST, 14:#CLO, 16:199, 18:1, 20:0, 22:0, 24:1, 25:NORMAL37
$BWDSTART = FALSE
LDAT_ACT=LL_OLP40
BAS(#CP_DAT)
FDAT_ACT=FSWP_60_9310
BAS(#FRAMES)
BAS(#VEL_CP,LL_OLP40.VEL)
S_ACT.GUN=3
S_ACT.PAIR=SDEFAULT.PAIR
S_ACT.RETR=#CLO
S_ACT.CLO_TM=1
S_ACT.PGNO1=199
S_ACT.PGNO2=SDEFAULT.PGNO2
S_ACT.PRESS1=SDEFAULT.PRESS1
S_ACT.PRESS2=SDEFAULT.PRESS2
S_READY=FALSE
LIN XSWP_60_9310
USERSPOT(#SPOT, S_ACT)
WAIT FOR S_READY
;ENDFOLD

;FOLD ; SWP_60_9312;%{PE}%R 4.1.16,%MKUKATPBASIS,%CCOMMENT,%VNORMAL,%P 2:SWP_60_9312
;ENDFOLD
;FOLD LIN SWP_60_9212 L_OLP41 SPOT Gun= 3 RETR CLS PgNo1= 199 ACTIVE= 1 Tool[3]:GUN C02 Base[3]:Atego/Axor;%{PE}%R 4.1.12,%MKUKATPSPOT,%CSPOT,%VLIN,%P 1:LIN, 2:SWP_60_9212, 3:, 5:2, 7:L_OLP41, 10:3, 12:#FIRST, 14:#CLO, 16:199, 18:1, 20:0, 22:0, 24:1, 25:NORMAL37
$BWDSTART = FALSE
LDAT_ACT=LL_OLP41
BAS(#CP_DAT)
FDAT_ACT=FSWP_60_9212
BAS(#FRAMES)
BAS(#VEL_CP,LL_OLP41.VEL)
S_ACT.GUN=3
S_ACT.PAIR=SDEFAULT.PAIR
S_ACT.RETR=#CLO
S_ACT.CLO_TM=1
S_ACT.PGNO1=199
S_ACT.PGNO2=SDEFAULT.PGNO2
S_ACT.PRESS1=SDEFAULT.PRESS1
S_ACT.PRESS2=SDEFAULT.PRESS2
S_READY=FALSE
LIN XSWP_60_9212
USERSPOT(#SPOT, S_ACT)
WAIT FOR S_READY
;ENDFOLD

;FOLD ; SWP_60_9250;%{PE}%R 4.1.16,%MKUKATPBASIS,%CCOMMENT,%VNORMAL,%P 2:SWP_60_9250
;ENDFOLD
;FOLD LIN SWP_60_9250 L_OLP42 SPOT Gun= 3 RETR CLS PgNo1= 199 ACTIVE= 1 Tool[3]:GUN C02 Base[3]:Atego/Axor;%{PE}%R 4.1.12,%MKUKATPSPOT,%CSPOT,%VLIN,%P 1:LIN, 2:SWP_60_9250, 3:, 5:2, 7:L_OLP42, 10:3, 12:#FIRST, 14:#CLO, 16:199, 18:1, 20:0, 22:0, 24:1, 25:NORMAL37
$BWDSTART = FALSE
LDAT_ACT=LL_OLP42
BAS(#CP_DAT)
FDAT_ACT=FSWP_60_9250
BAS(#FRAMES)
BAS(#VEL_CP,LL_OLP42.VEL)
S_ACT.GUN=3
S_ACT.PAIR=SDEFAULT.PAIR
S_ACT.RETR=#CLO
S_ACT.CLO_TM=1
S_ACT.PGNO1=199
S_ACT.PGNO2=SDEFAULT.PGNO2
S_ACT.PRESS1=SDEFAULT.PRESS1
S_ACT.PRESS2=SDEFAULT.PRESS2
S_READY=FALSE
LIN XSWP_60_9250
USERSPOT(#SPOT, S_ACT)
WAIT FOR S_READY
;ENDFOLD

;FOLD ; SWP_60_9248;%{PE}%R 4.1.16,%MKUKATPBASIS,%CCOMMENT,%VNORMAL,%P 2:SWP_60_9248
;ENDFOLD
;FOLD LIN SWP_60_9248 L_OLP43 SPOT Gun= 3 RETR CLS PgNo1= 199 ACTIVE= 1 Tool[3]:GUN C02 Base[3]:Atego/Axor;%{PE}%R 4.1.12,%MKUKATPSPOT,%CSPOT,%VLIN,%P 1:LIN, 2:SWP_60_9248, 3:, 5:2, 7:L_OLP43, 10:3, 12:#FIRST, 14:#CLO, 16:199, 18:1, 20:0, 22:0, 24:1, 25:NORMAL37
$BWDSTART = FALSE
LDAT_ACT=LL_OLP43
BAS(#CP_DAT)
FDAT_ACT=FSWP_60_9248
BAS(#FRAMES)
BAS(#VEL_CP,LL_OLP43.VEL)
S_ACT.GUN=3
S_ACT.PAIR=SDEFAULT.PAIR
S_ACT.RETR=#CLO
S_ACT.CLO_TM=1
S_ACT.PGNO1=199
S_ACT.PGNO2=SDEFAULT.PGNO2
S_ACT.PRESS1=SDEFAULT.PRESS1
S_ACT.PRESS2=SDEFAULT.PRESS2
S_READY=FALSE
LIN XSWP_60_9248
USERSPOT(#SPOT, S_ACT)
WAIT FOR S_READY
;ENDFOLD

;FOLD ; SWP_60_9246;%{PE}%R 4.1.16,%MKUKATPBASIS,%CCOMMENT,%VNORMAL,%P 2:SWP_60_9246
;ENDFOLD
;FOLD LIN SWP_60_9246 L_OLP44 SPOT Gun= 3 RETR CLS PgNo1= 199 ACTIVE= 1 Tool[3]:GUN C02 Base[3]:Atego/Axor;%{PE}%R 4.1.12,%MKUKATPSPOT,%CSPOT,%VLIN,%P 1:LIN, 2:SWP_60_9246, 3:, 5:2, 7:L_OLP44, 10:3, 12:#FIRST, 14:#CLO, 16:199, 18:1, 20:0, 22:0, 24:1, 25:NORMAL37
$BWDSTART = FALSE
LDAT_ACT=LL_OLP44
BAS(#CP_DAT)
FDAT_ACT=FSWP_60_9246
BAS(#FRAMES)
BAS(#VEL_CP,LL_OLP44.VEL)
S_ACT.GUN=3
S_ACT.PAIR=SDEFAULT.PAIR
S_ACT.RETR=#CLO
S_ACT.CLO_TM=1
S_ACT.PGNO1=199
S_ACT.PGNO2=SDEFAULT.PGNO2
S_ACT.PRESS1=SDEFAULT.PRESS1
S_ACT.PRESS2=SDEFAULT.PRESS2
S_READY=FALSE
LIN XSWP_60_9246
USERSPOT(#SPOT, S_ACT)
WAIT FOR S_READY
;ENDFOLD

;FOLD ; SWP_60_9244;%{PE}%R 4.1.16,%MKUKATPBASIS,%CCOMMENT,%VNORMAL,%P 2:SWP_60_9244
;ENDFOLD
;FOLD LIN SWP_60_9244 L_OLP45 SPOT Gun= 3 RETR CLS PgNo1= 199 ACTIVE= 1 Tool[3]:GUN C02 Base[3]:Atego/Axor;%{PE}%R 4.1.12,%MKUKATPSPOT,%CSPOT,%VLIN,%P 1:LIN, 2:SWP_60_9244, 3:, 5:2, 7:L_OLP45, 10:3, 12:#FIRST, 14:#CLO, 16:199, 18:1, 20:0, 22:0, 24:1, 25:NORMAL37
$BWDSTART = FALSE
LDAT_ACT=LL_OLP45
BAS(#CP_DAT)
FDAT_ACT=FSWP_60_9244
BAS(#FRAMES)
BAS(#VEL_CP,LL_OLP45.VEL)
S_ACT.GUN=3
S_ACT.PAIR=SDEFAULT.PAIR
S_ACT.RETR=#CLO
S_ACT.CLO_TM=1
S_ACT.PGNO1=199
S_ACT.PGNO2=SDEFAULT.PGNO2
S_ACT.PRESS1=SDEFAULT.PRESS1
S_ACT.PRESS2=SDEFAULT.PRESS2
S_READY=FALSE
LIN XSWP_60_9244
USERSPOT(#SPOT, S_ACT)
WAIT FOR S_READY
;ENDFOLD

;FOLD ; SWP_60_9242;%{PE}%R 4.1.16,%MKUKATPBASIS,%CCOMMENT,%VNORMAL,%P 2:SWP_60_9242
;ENDFOLD
;FOLD LIN SWP_60_9242 L_OLP46 SPOT Gun= 3 RETR CLS PgNo1= 199 ACTIVE= 1 Tool[3]:GUN C02 Base[3]:Atego/Axor;%{PE}%R 4.1.12,%MKUKATPSPOT,%CSPOT,%VLIN,%P 1:LIN, 2:SWP_60_9242, 3:, 5:2, 7:L_OLP46, 10:3, 12:#FIRST, 14:#CLO, 16:199, 18:1, 20:0, 22:0, 24:1, 25:NORMAL37
$BWDSTART = FALSE
LDAT_ACT=LL_OLP46
BAS(#CP_DAT)
FDAT_ACT=FSWP_60_9242
BAS(#FRAMES)
BAS(#VEL_CP,LL_OLP46.VEL)
S_ACT.GUN=3
S_ACT.PAIR=SDEFAULT.PAIR
S_ACT.RETR=#CLO
S_ACT.CLO_TM=1
S_ACT.PGNO1=199
S_ACT.PGNO2=SDEFAULT.PGNO2
S_ACT.PRESS1=SDEFAULT.PRESS1
S_ACT.PRESS2=SDEFAULT.PRESS2
S_READY=FALSE
LIN XSWP_60_9242
USERSPOT(#SPOT, S_ACT)
WAIT FOR S_READY
;ENDFOLD

;FOLD ; SWP_60_9240;%{PE}%R 4.1.16,%MKUKATPBASIS,%CCOMMENT,%VNORMAL,%P 2:SWP_60_9240
;ENDFOLD
;FOLD LIN SWP_60_9240 L_OLP47 SPOT Gun= 3 RETR CLS PgNo1= 199 ACTIVE= 1 Tool[3]:GUN C02 Base[3]:Atego/Axor;%{PE}%R 4.1.12,%MKUKATPSPOT,%CSPOT,%VLIN,%P 1:LIN, 2:SWP_60_9240, 3:, 5:2, 7:L_OLP47, 10:3, 12:#FIRST, 14:#CLO, 16:199, 18:1, 20:0, 22:0, 24:1, 25:NORMAL37
$BWDSTART = FALSE
LDAT_ACT=LL_OLP47
BAS(#CP_DAT)
FDAT_ACT=FSWP_60_9240
BAS(#FRAMES)
BAS(#VEL_CP,LL_OLP47.VEL)
S_ACT.GUN=3
S_ACT.PAIR=SDEFAULT.PAIR
S_ACT.RETR=#CLO
S_ACT.CLO_TM=1
S_ACT.PGNO1=199
S_ACT.PGNO2=SDEFAULT.PGNO2
S_ACT.PRESS1=SDEFAULT.PRESS1
S_ACT.PRESS2=SDEFAULT.PRESS2
S_READY=FALSE
LIN XSWP_60_9240
USERSPOT(#SPOT, S_ACT)
WAIT FOR S_READY
;ENDFOLD

;FOLD ; SWP_60_9238;%{PE}%R 4.1.16,%MKUKATPBASIS,%CCOMMENT,%VNORMAL,%P 2:SWP_60_9238
;ENDFOLD
;FOLD LIN SWP_60_9238 L_OLP48 SPOT Gun= 3 RETR CLS PgNo1= 199 ACTIVE= 1 Tool[3]:GUN C02 Base[3]:Atego/Axor;%{PE}%R 4.1.12,%MKUKATPSPOT,%CSPOT,%VLIN,%P 1:LIN, 2:SWP_60_9238, 3:, 5:2, 7:L_OLP48, 10:3, 12:#FIRST, 14:#CLO, 16:199, 18:1, 20:0, 22:0, 24:1, 25:NORMAL37
$BWDSTART = FALSE
LDAT_ACT=LL_OLP48
BAS(#CP_DAT)
FDAT_ACT=FSWP_60_9238
BAS(#FRAMES)
BAS(#VEL_CP,LL_OLP48.VEL)
S_ACT.GUN=3
S_ACT.PAIR=SDEFAULT.PAIR
S_ACT.RETR=#CLO
S_ACT.CLO_TM=1
S_ACT.PGNO1=199
S_ACT.PGNO2=SDEFAULT.PGNO2
S_ACT.PRESS1=SDEFAULT.PRESS1
S_ACT.PRESS2=SDEFAULT.PRESS2
S_READY=FALSE
LIN XSWP_60_9238
USERSPOT(#SPOT, S_ACT)
WAIT FOR S_READY
;ENDFOLD

;FOLD ; SWP_60_9236;%{PE}%R 4.1.16,%MKUKATPBASIS,%CCOMMENT,%VNORMAL,%P 2:SWP_60_9236
;ENDFOLD
;FOLD LIN SWP_60_9236 L_OLP49 SPOT Gun= 3 RETR OPN PgNo1= 199 ACTIVE= 1 Tool[3]:GUN C02 Base[3]:Atego/Axor;%{PE}%R 4.1.12,%MKUKATPSPOT,%CSPOT,%VLIN,%P 1:LIN, 2:SWP_60_9236, 3:, 5:2, 7:L_OLP49, 10:3, 12:#FIRST, 14:#OPN, 16:199, 18:1, 20:0, 22:0, 24:1, 25:NORMAL37
$BWDSTART = FALSE
LDAT_ACT=LL_OLP49
BAS(#CP_DAT)
FDAT_ACT=FSWP_60_9236
BAS(#FRAMES)
BAS(#VEL_CP,LL_OLP49.VEL)
S_ACT.GUN=3
S_ACT.PAIR=SDEFAULT.PAIR
S_ACT.RETR=#OPN
S_ACT.CLO_TM=1
S_ACT.PGNO1=199
S_ACT.PGNO2=SDEFAULT.PGNO2
S_ACT.PRESS1=SDEFAULT.PRESS1
S_ACT.PRESS2=SDEFAULT.PRESS2
S_READY=FALSE
LIN XSWP_60_9236
USERSPOT(#SPOT, S_ACT)
WAIT FOR S_READY
;ENDFOLD

;FOLD LIN SWP_60_9234 CPDAT30 SPOT Gun= 3 RETR OPN PgNo1= 197 ACTIVE= 1 Tool[3]:GUN C02 Base[3]:Atego/Axor;%{PE}%R 4.1.12,%MKUKATPSPOT,%CSPOT,%VLIN,%P 1:LIN, 2:SWP_60_9234, 3:, 5:2, 7:CPDAT30, 10:3, 12:#FIRST, 14:#OPN, 16:197, 18:1, 20:0, 22:0, 24:1, 25:NORMAL
$BWDSTART = FALSE
LDAT_ACT=LCPDAT30
BAS(#CP_DAT)
FDAT_ACT=FSWP_60_9234
BAS(#FRAMES)
BAS(#VEL_CP,LCPDAT30.VEL)
S_ACT.GUN=3
S_ACT.PAIR=SDEFAULT.PAIR
S_ACT.RETR=#OPN
S_ACT.CLO_TM=1
S_ACT.PGNO1=197
S_ACT.PGNO2=SDEFAULT.PGNO2
S_ACT.PRESS1=SDEFAULT.PRESS1
S_ACT.PRESS2=SDEFAULT.PRESS2
S_READY=FALSE
LIN XSWP_60_9234
USERSPOT(#SPOT, S_ACT)
WAIT FOR S_READY
;ENDFOLD


;FOLD PTP P23 CONT Vel= 100 % PDAT13 Tool[1]:GUN C1 Base[3]:Atego/Axor;%{PE}%R 4.1.16,%MKUKATPBASIS,%CMOVE,%VPTP,%P 1:PTP, 2:P23, 3:C_PTP, 5:100, 7:PDAT13
$BWDSTART = FALSE
PDAT_ACT=PPDAT13
BAS(#PTP_DAT)
FDAT_ACT=FP23
BAS(#FRAMES)
BAS(#VEL_PTP,100)
PTP XP23 C_PTP
;ENDFOLD
;FOLD PTP P22 CONT Vel= 100 % PDAT12 Tool[1]:GUN C1 Base[3]:Atego/Axor;%{PE}%R 4.1.16,%MKUKATPBASIS,%CMOVE,%VPTP,%P 1:PTP, 2:P22, 3:C_PTP, 5:100, 7:PDAT12
$BWDSTART = FALSE
PDAT_ACT=PPDAT12
BAS(#PTP_DAT)
FDAT_ACT=FP22
BAS(#FRAMES)
BAS(#VEL_PTP,100)
PTP XP22 C_PTP
;ENDFOLD
;FOLD PTP P21 CONT Vel= 100 % PDAT11 Tool[1]:GUN C1 Base[3]:Atego/Axor;%{PE}%R 4.1.16,%MKUKATPBASIS,%CMOVE,%VPTP,%P 1:PTP, 2:P21, 3:C_PTP, 5:100, 7:PDAT11
$BWDSTART = FALSE
PDAT_ACT=PPDAT11
BAS(#PTP_DAT)
FDAT_ACT=FP21
BAS(#FRAMES)
BAS(#VEL_PTP,100)
PTP XP21 C_PTP
;ENDFOLD




;FOLD PTP l091 CONT Vel= 100 % P_OLP50 Tool[3] Base[3]:Atego/Axor;%{PE}%R 4.1.16,%MKUKATPBASIS,%CMOVE,%VPTP,%P 1:PTP, 2:l091, 3:C_PTP, 5:100, 7:P_OLP50
$BWDSTART = FALSE
PDAT_ACT=PP_OLP50
BAS(#PTP_DAT)
FDAT_ACT=Fl091
BAS(#FRAMES)
BAS(#VEL_PTP,100)
PTP Xl091 C_PTP
;ENDFOLD
;FOLD PTP l096 CONT Vel= 100 % P_OLP51 Tool[3] Base[3]:Atego/Axor;%{PE}%R 4.1.16,%MKUKATPBASIS,%CMOVE,%VPTP,%P 1:PTP, 2:l096, 3:C_PTP, 5:100, 7:P_OLP51
$BWDSTART = FALSE
PDAT_ACT=PP_OLP51
BAS(#PTP_DAT)
FDAT_ACT=Fl096
BAS(#FRAMES)
BAS(#VEL_PTP,100)
PTP Xl096 C_PTP
;ENDFOLD

;FOLD PTP PS_32 CONT Vel= 100 % PDAT26 Tool[3]:GUN C02 Base[3]:Atego/Axor;%{PE}%R 4.1.16,%MKUKATPBASIS,%CMOVE,%VPTP,%P 1:PTP, 2:PS_32, 3:C_PTP, 5:100, 7:PDAT26
$BWDSTART = FALSE
PDAT_ACT=PPDAT26
BAS(#PTP_DAT)
FDAT_ACT=FPS_32
BAS(#FRAMES)
BAS(#VEL_PTP,100)
PTP XPS_32 C_PTP
;ENDFOLD

;FOLD ; Desliga Intertravamento 7 c/ R03 Pinca C02;%{PE}%R 4.1.16,%MKUKATPBASIS,%CCOMMENT,%VNORMAL,%P 2:Desliga Intertravamento 7 c/ R03 Pinca C02
;ENDFOLD

;FOLD Kollision.Monitoring_AREA_1_Off ;%{PE}%MKUKATPUSER
COLLSTOP( 7, 2 )
;ENDFOLD

;FOLD PTP P6 CONT Vel= 100 % PDAT6 Tool[3]:GUN C02 Base[3]:Atego/Axor;%{PE}%R 4.1.16,%MKUKATPBASIS,%CMOVE,%VPTP,%P 1:PTP, 2:P6, 3:C_PTP, 5:100, 7:PDAT6
$BWDSTART = FALSE
PDAT_ACT=PPDAT6
BAS(#PTP_DAT)
FDAT_ACT=FP6
BAS(#FRAMES)
BAS(#VEL_PTP,100)
PTP XP6 C_PTP
;ENDFOLD

;FOLD ; Desliga Intertravamento 1 c/ R01;%{PE}%R 4.1.16,%MKUKATPBASIS,%CCOMMENT,%VNORMAL,%P 2:Desliga Intertravamento 1 c/ R01
;ENDFOLD
;FOLD ; Desliga Intertravamento 8 c/ R03 Pinca C01;%{PE}%R 4.1.16,%MKUKATPBASIS,%CCOMMENT,%VNORMAL,%P 2:Desliga Intertravamento 8 c/ R03 Pinca C01
;ENDFOLD
;FOLD ; Desliga Intertravamento 10 c/ R02;%{PE}%R 4.1.16,%MKUKATPBASIS,%CCOMMENT,%VNORMAL,%P 2:Desliga Intertravamento 10 c/ R02
;ENDFOLD
;FOLD Kollision.Ueberwachung_1_Aus ;%{PE}%MKUKATPUSER
COLLSTOP( 1, 2 )
;ENDFOLD
;FOLD Kollision.Monitoring_AREA_2_Off ;%{PE}%MKUKATPUSER
COLLSTOP( 8, 2 )
;ENDFOLD
;FOLD Kollision.Monitoring_AREA_4_Off ;%{PE}%MKUKATPUSER
COLLSTOP( 10, 2 )
;ENDFOLD

;FOLD ; Desliga Intertravamento 3 c/ R03;%{PE}%R 4.1.16,%MKUKATPBASIS,%CCOMMENT,%VNORMAL,%P 2:Desliga Intertravamento 7 c/ R03
;ENDFOLD
;FOLD Kollision.Ueberwachung_3_Aus ;%{PE}%MKUKATPUSER
COLLSTOP( 3, 2 )
;ENDFOLD

IF (NOT(GHOST())) THEN
IF FraesAnf(3) THEN
f_Fraes3()
ENDIF
ENDIF

;FOLD PTP P24  Vel= 100 % PDAT19 Tool[3]:GUN C02 Base[0];%{PE}%R 4.1.16,%MKUKATPBASIS,%CMOVE,%VPTP,%P 1:PTP, 2:P24, 3:, 5:100, 7:PDAT19
$BWDSTART = FALSE
PDAT_ACT=PPDAT19
BAS(#PTP_DAT)
FDAT_ACT=FP24
BAS(#FRAMES)
BAS(#VEL_PTP,100)
PTP XP24
;ENDFOLD

end_weld ( )
END

--- ps_b_ltb_res_c02.dat ---
&ACCESS RVO1
&COMMENT Solda Axor LTB
DEFDAT ps_b_ltb_res_c02
;FOLD EXTERNAL DECLARATIONS;%{PE}%V2.2.2,%MKUKATPBASIS,%CEXT,%VCOMMON,%P
;FOLD BAS EXT;%{PE}%V2.2.2,%MKUKATPBASIS,%CEXT,%VEXT,%P
EXT  BAS (BAS_COMMAND  :IN,REAL  :IN )
DECL INT SUCCESS
;ENDFOLD
;FOLD A10 EXT;%{E}%V2.2.2,%MKUKATPARC,%CEXT,%VEXT,%P
EXT  A10 (A_CMD_T  :IN,A_STRT_T  :IN,A_WELD_T  :IN,A_END_T  :IN,INT  :IN )
;ENDFOLD
;FOLD A20 EXT;%{E}%V2.2.2,%MKUKATPA20,%CEXT,%VEXT,%P
EXT  A20 (INT  :IN,WELD_ST  :IN,WELD_FI  :IN,INT  :IN )
;ENDFOLD
;FOLD GRIPPER EXT;%{E}%V2.2.2,%MKUKATPGRIPPER,%CEXT,%VEXT,%P
EXT  H50 (INT  :IN,INT  :IN,INT  :IN,GRP_TYP  :IN )
;ENDFOLD
;FOLD SPOT EXT;%{E}%V2.2.2,%MKUKATPSPOT,%CEXT,%VEXT,%P
EXT  USERSPOT (S_COMMAND  :IN,SPOT_TYPE  :IN )
;ENDFOLD
;FOLD TOUCHSENSE EXT;%{E}%V2.2.2,%MKUKATPTS,%CEXT,%VEXT,%P
EXT  H70 (INT  :IN,SRCH_TYP_2  :OUT,E6POS  :IN,SRCH_TYP_3  :IN,SRCH_TYP_2  :IN,SRCH_TYP_2  :IN,SRCH_TYP_2  :IN,SRCH_TYP_2  :IN,SRCH_TYP_2  :IN,INT  :IN )
;ENDFOLD
;FOLD USER EXT;%{}%V2.2.2,%MKUKATPUSER,%CEXT,%VEXT,%P
;Make here your modifications
;ENDFOLD
;ENDFOLD

DECL FDAT Fl005={TOOL_NO 3,BASE_NO 3,IPO_FRAME #BASE}
DECL PDAT PP_OLP2={VEL 100.0,ACC 100.0,APO_DIST 0.0}
DECL E6POS Xl005={x -259.953003,y 860.291992,z 674.213013,a 106.465103,b 65.7322998,c -50.9701004,s 2,t 42}
DECL FDAT Fl010={TOOL_NO 3,BASE_NO 3,IPO_FRAME #BASE}
DECL PDAT PP_OLP3={VEL 100.0,ACC 100.0,APO_DIST 0.0}
DECL E6POS Xl010={x 238.578995,y 878.294983,z 634.81897,a 106.465103,b 65.7322998,c -50.9701004,s 2,t 43}
DECL FDAT Fl015={TOOL_NO 3,BASE_NO 3,IPO_FRAME #BASE}
DECL PDAT PP_OLP4={VEL 100.0,ACC 100.0,APO_DIST 0.0}
DECL E6POS Xl015={x 233.995102,y 927.062683,z 508.398987,a 106.4627,b 65.7314301,c -48.9741592,s 2,t 43,e1 0.0,e2 0.0,e3 0.0,e4 0.0,e5 0.0,e6 0.0}
DECL LDAT LL_OLP1={VEL 2.0,ACC 100.0,APO_DIST 0.0,APO_FAC 0.0}
DECL FDAT Fl020={TOOL_NO 3,BASE_NO 3,IPO_FRAME #BASE}
DECL PDAT PP_OLP5={VEL 100.0,ACC 100.0,APO_DIST 0.0}
DECL E6POS Xl020={x 240.050705,y 924.635925,z 506.612305,a 106.462997,b 65.7332382,c -48.9725304,s 2,t 43,e1 0.0,e2 0.0,e3 0.0,e4 0.0,e5 0.0,e6 0.0}
DECL FDAT Fl025={TOOL_NO 3,BASE_NO 3,IPO_FRAME #BASE}
DECL PDAT PP_OLP6={VEL 100.0,ACC 100.0,APO_DIST 0.0}
DECL E6POS Xl025={x 230.037399,y 926.909119,z 610.785889,a 106.4646,b 65.7323837,c -48.9705811,s 2,t 43,e1 0.0,e2 0.0,e3 0.0,e4 0.0,e5 0.0,e6 0.0}
DECL FDAT Fl030={TOOL_NO 3,BASE_NO 3,IPO_FRAME #BASE}
DECL PDAT PP_OLP7={VEL 100.0,ACC 100.0,APO_DIST 0.0}
DECL E6POS Xl030={x 193.569397,y 878.43573,z 618.731201,a 136.368896,b 76.3886337,c -42.6437798,s 2,t 43,e1 0.0,e2 0.0,e3 0.0,e4 0.0,e5 0.0,e6 0.0}
DECL E6POS Xl011={x 216.297104,y 817.987915,z 621.025818,a -90.0010071,b 86.8945236,c 89.9989166,s 2,t 43,e1 0.0,e2 0.0,e3 0.0,e4 0.0,e5 0.0,e6 0.0}
DECL FDAT Fl011={TOOL_NO 3,BASE_NO 3,IPO_FRAME #BASE}
DECL PDAT PP_OLP11={VEL 100.0,ACC 100.0,APO_DIST 0.0}
DECL E6POS Xl016={x 210.0,y 837.984985,z 424.028992,a -89.9999008,b 86.8943024,c 90.0000992,s 2,t 43}
DECL FDAT Fl016={TOOL_NO 3,BASE_NO 3,IPO_FRAME #BASE}
DECL PDAT PP_OLP12={VEL 100.0,ACC 100.0,APO_DIST 0.0}
DECL E6POS XSWP_60_7354={x 203.809906,y 837.713989,z 419.105103,a -90.024231,b 86.8921432,c 89.974617,s 2,t 43,e1 0.0,e2 0.0,e3 0.0,e4 0.0,e5 0.0,e6 0.0}
DECL FDAT FSWP_60_7354={TOOL_NO 3,BASE_NO 3,IPO_FRAME #BASE}
DECL LDAT LL_OLP2={VEL 2.0,ACC 100.0,APO_DIST 0.0,APO_FAC 0.0}
DECL E6POS XSWP_60_7356={x 204.900299,y 813.062012,z 427.303589,a -90.0252304,b 86.8959122,c 89.9749298,s 2,t 43,e1 0.0,e2 0.0,e3 0.0,e4 0.0,e5 0.0,e6 0.0}
DECL FDAT FSWP_60_7356={TOOL_NO 3,BASE_NO 3,IPO_FRAME #BASE}
DECL LDAT LL_OLP3={VEL 2.0,ACC 100.0,APO_DIST 0.0,APO_FAC 0.0}
DECL E6POS XSWP_60_7358={x 205.666595,y 785.228699,z 444.857788,a -90.0419312,b 86.8953781,c 89.9582901,s 2,t 43,e1 0.0,e2 0.0,e3 0.0,e4 0.0,e5 0.0,e6 0.0}
DECL FDAT FSWP_60_7358={TOOL_NO 3,BASE_NO 3,IPO_FRAME #BASE}
DECL LDAT LL_OLP4={VEL 2.0,ACC 100.0,APO_DIST 0.0,APO_FAC 0.0}
DECL E6POS XSWP_60_7360={x 203.261703,y 756.455627,z 466.485809,a -89.9985809,b 86.8937683,c 90.0012436,s 2,t 43,e1 0.0,e2 0.0,e3 0.0,e4 0.0,e5 0.0,e6 0.0}
DECL FDAT FSWP_60_7360={TOOL_NO 3,BASE_NO 3,IPO_FRAME #BASE}
DECL LDAT LL_OLP5={VEL 2.0,ACC 100.0,APO_DIST 0.0,APO_FAC 0.0}
DECL E6POS XSWP_60_7362={x 206.944794,y 725.337585,z 475.673492,a 89.9988937,b 70.9206924,c -90.0019226,s 2,t 43,e1 0.0,e2 0.0,e3 0.0,e4 0.0,e5 0.0,e6 0.0}
DECL FDAT FSWP_60_7362={TOOL_NO 3,BASE_NO 3,IPO_FRAME #BASE}
DECL LDAT LL_OLP6={VEL 2.0,ACC 100.0,APO_DIST 0.0,APO_FAC 0.0}
DECL E6POS XSWP_60_7364={x 206.622696,y 692.928894,z 476.588287,a -90.0024414,b 86.1575623,c 89.9975586,s 2,t 43,e1 0.0,e2 0.0,e3 0.0,e4 0.0,e5 0.0,e6 0.0}
DECL FDAT FSWP_60_7364={TOOL_NO 3,BASE_NO 3,IPO_FRAME #BASE}
DECL LDAT LL_OLP7={VEL 2.0,ACC 100.0,APO_DIST 0.0,APO_FAC 0.0}
DECL E6POS XSWP_60_7366={x 203.315002,y 660.348389,z 476.359894,a -90.0006638,b 56.1120415,c 89.9992981,s 2,t 43,e1 0.0,e2 0.0,e3 0.0,e4 0.0,e5 0.0,e6 0.0}
DECL FDAT FSWP_60_7366={TOOL_NO 3,BASE_NO 3,IPO_FRAME #BASE}
DECL LDAT LL_OLP8={VEL 2.0,ACC 100.0,APO_DIST 0.0,APO_FAC 0.0}
DECL E6POS XSWP_60_7368={x 206.116501,y 634.32843,z 476.098907,a -90.0014801,b 58.2454681,c 90.0003967,s 2,t 43,e1 0.0,e2 0.0,e3 0.0,e4 0.0,e5 0.0,e6 0.0}
DECL FDAT FSWP_60_7368={TOOL_NO 3,BASE_NO 3,IPO_FRAME #BASE}
DECL LDAT LL_OLP9={VEL 2.0,ACC 100.0,APO_DIST 0.0,APO_FAC 0.0}
DECL E6POS XSWP_60_7370={x 205.649307,y 608.364075,z 476.227295,a -90.000618,b 59.0425911,c 89.9998627,s 2,t 43,e1 0.0,e2 0.0,e3 0.0,e4 0.0,e5 0.0,e6 0.0}
DECL FDAT FSWP_60_7370={TOOL_NO 3,BASE_NO 3,IPO_FRAME #BASE}
DECL LDAT LL_OLP10={VEL 2.0,ACC 100.0,APO_DIST 0.0,APO_FAC 0.0}
DECL E6POS XSWP_60_7372={x 207.227097,y 582.377502,z 476.378601,a -90.0000229,b 59.7199898,c 90.0000229,s 2,t 43,e1 0.0,e2 0.0,e3 0.0,e4 0.0,e5 0.0,e6 0.0}
DECL FDAT FSWP_60_7372={TOOL_NO 3,BASE_NO 3,IPO_FRAME #BASE}
DECL LDAT LL_OLP11={VEL 2.0,ACC 100.0,APO_DIST 0.0,APO_FAC 0.0}
DECL E6POS XSWP_60_7374={x 206.739594,y 556.385376,z 476.24881,a -89.9996872,b 60.0724792,c 89.9999695,s 2,t 43,e1 0.0,e2 0.0,e3 0.0,e4 0.0,e5 0.0,e6 0.0}
DECL FDAT FSWP_60_7374={TOOL_NO 3,BASE_NO 3,IPO_FRAME #BASE}
DECL LDAT LL_OLP12={VEL 2.0,ACC 100.0,APO_DIST 0.0,APO_FAC 0.0}
DECL E6POS Xl026={x 232.763107,y 556.379089,z 476.253387,a -89.9998627,b 59.855629,c 90.0001068,s 2,t 43,e1 0.0,e2 0.0,e3 0.0,e4 0.0,e5 0.0,e6 0.0}
DECL FDAT Fl026={TOOL_NO 3,BASE_NO 3,IPO_FRAME #BASE}
DECL PDAT PP_OLP14={VEL 100.0,ACC 100.0,APO_DIST 0.0}
DECL E6POS Xl031={x 234.033997,y 429.904907,z 476.388092,a -90.0016632,b 59.8551102,c 89.9992065,s 2,t 43,e1 0.0,e2 0.0,e3 0.0,e4 0.0,e5 0.0,e6 0.0}
DECL FDAT Fl031={TOOL_NO 3,BASE_NO 3,IPO_FRAME #BASE}
DECL PDAT PP_OLP15={VEL 100.0,ACC 100.0,APO_DIST 0.0}
DECL E6POS XSWP_60_7376={x 205.848206,y 441.043304,z 482.712006,a -89.9979706,b 60.0047493,c 90.0008774,s 2,t 43,e1 0.0,e2 0.0,e3 0.0,e4 0.0,e5 0.0,e6 0.0}
DECL FDAT FSWP_60_7376={TOOL_NO 3,BASE_NO 3,IPO_FRAME #BASE}
DECL LDAT LL_OLP13={VEL 2.0,ACC 100.0,APO_DIST 0.0,APO_FAC 0.0}
DECL E6POS XSWP_60_7378={x 206.973907,y 431.014099,z 441.041809,a -89.9991226,b 61.5301018,c 90.0008698,s 2,t 43,e1 0.0,e2 0.0,e3 0.0,e4 0.0,e5 0.0,e6 0.0}
DECL FDAT FSWP_60_7378={TOOL_NO 3,BASE_NO 3,IPO_FRAME #BASE}
DECL LDAT LL_OLP14={VEL 2.0,ACC 100.0,APO_DIST 0.0,APO_FAC 0.0}
DECL E6POS XSWP_60_7380={x 206.840393,y 416.639099,z 400.304108,a -89.9998703,b 62.6937904,c 90.0006027,s 2,t 43,e1 0.0,e2 0.0,e3 0.0,e4 0.0,e5 0.0,e6 0.0}
DECL FDAT FSWP_60_7380={TOOL_NO 3,BASE_NO 3,IPO_FRAME #BASE}
DECL LDAT LL_OLP15={VEL 2.0,ACC 100.0,APO_DIST 0.0,APO_FAC 0.0}
DECL E6POS XSWP_60_7220={x 205.599396,y 39.2980804,z 386.423615,a -89.9959183,b 44.4748917,c 89.9934921,s 2,t 43,e1 0.0,e2 0.0,e3 0.0,e4 0.0,e5 0.0,e6 0.0}
DECL FDAT FSWP_60_7220={TOOL_NO 3,BASE_NO 3,IPO_FRAME #BASE}
DECL E6POS XSWP_60_7222={x 206.282593,y 88.0883484,z 386.359711,a -89.9976273,b 44.4760399,c 89.9922333,s 2,t 43,e1 0.0,e2 0.0,e3 0.0,e4 0.0,e5 0.0,e6 0.0}
DECL FDAT FSWP_60_7222={TOOL_NO 3,BASE_NO 3,IPO_FRAME #BASE}
DECL LDAT LL_OLP31={VEL 2.0,ACC 50.0,APO_DIST 0.0,APO_FAC 0.0}
DECL LDAT LL_OLP32={VEL 2.0,ACC 50.0,APO_DIST 0.0,APO_FAC 0.0}
DECL LDAT LL_OLP33={VEL 2.0,ACC 100.0,APO_DIST 0.0,APO_FAC 0.0}
DECL LDAT LL_OLP34={VEL 2.0,ACC 100.0,APO_DIST 0.0,APO_FAC 0.0}
DECL E6POS XSWP_60_7260={x 181.102097,y 50.2497406,z 492.070099,a -80.3131027,b 32.1295509,c 107.793098,s 2,t 11,e1 0.0,e2 0.0,e3 0.0,e4 0.0,e5 0.0,e6 0.0}
DECL FDAT FSWP_60_7260={TOOL_NO 3,BASE_NO 3,IPO_FRAME #BASE}
DECL E6POS XSWP_60_7261={x 180.671097,y 1.26443899,z 490.916901,a -80.5087128,b 31.6135597,c 107.6959,s 2,t 11,e1 0.0,e2 0.0,e3 0.0,e4 0.0,e5 0.0,e6 0.0}
DECL FDAT FSWP_60_7261={TOOL_NO 3,BASE_NO 3,IPO_FRAME #BASE}
DECL LDAT LL_OLP36={VEL 2.0,ACC 100.0,APO_DIST 0.0,APO_FAC 0.0}
DECL LDAT LL_OLP37={VEL 2.0,ACC 100.0,APO_DIST 0.0,APO_FAC 0.0}
DECL LDAT LL_OLP38={VEL 2.0,ACC 100.0,APO_DIST 0.0,APO_FAC 0.0}
DECL E6POS Xl086={x 160.914307,y 87.6342468,z 584.528687,a -71.1530838,b 50.3254509,c 113.916496,s 2,t 43,e1 0.0,e2 0.0,e3 0.0,e4 0.0,e5 0.0,e6 0.0}
DECL FDAT Fl086={TOOL_NO 3,BASE_NO 3,IPO_FRAME #BASE}
DECL PDAT PP_OLP49={VEL 100.0,ACC 100.0,APO_DIST 0.0}
DECL E6POS Xl091={x 172.296906,y 391.390808,z 683.738708,a -90.0011826,b 46.4089699,c 90.0007324,s 2,t 43,e1 0.0,e2 0.0,e3 0.0,e4 0.0,e5 0.0,e6 0.0}
DECL FDAT Fl091={TOOL_NO 3,BASE_NO 3,IPO_FRAME #BASE}
DECL PDAT PP_OLP50={VEL 100.0,ACC 100.0,APO_DIST 0.0}
DECL E6POS Xl096={x -352.044708,y 791.362305,z 674.194885,a 102.528297,b 65.7295227,c -50.9826317,s 2,t 42,e1 0.0,e2 0.0,e3 0.0,e4 0.0,e5 0.0,e6 0.0}
DECL FDAT Fl096={TOOL_NO 3,BASE_NO 3,IPO_FRAME #BASE}
DECL PDAT PP_OLP51={VEL 100.0,ACC 100.0,APO_DIST 0.0}
DECL E6POS XSWP_60_9320={x 232.712296,y 933.30603,z 511.6586,a 106.517799,b 65.743103,c -48.8957405,s 2,t 43,e1 0.0,e2 0.0,e3 0.0,e4 0.0,e5 0.0,e6 0.0}
DECL FDAT FSWP_60_9320={TOOL_NO 3,BASE_NO 3,IPO_FRAME #BASE}
DECL E6POS XP6={x -1383.52795,y 1084.21204,z 300.229401,a 152.116806,b 8.17701721,c 8.23256302,s 2,t 42,e1 0.0,e2 0.0,e3 0.0,e4 0.0,e5 0.0,e6 0.0}
DECL FDAT FP6={TOOL_NO 3,BASE_NO 3,IPO_FRAME #BASE}
DECL PDAT PPDAT6={VEL 100.0,ACC 100.0,APO_DIST 0.0}
DECL E6POS XP7={x 211.5793,y 905.759277,z 610.608276,a 118.261002,b 68.8623581,c -44.6343498,s 2,t 43,e1 0.0,e2 0.0,e3 0.0,e4 0.0,e5 0.0,e6 0.0}
DECL FDAT FP7={TOOL_NO 3,BASE_NO 3,IPO_FRAME #BASE}
DECL PDAT PPDAT7={VEL 100.0,ACC 100.0,APO_DIST 0.0}
DECL SPOT_SUGG_T LAST_SPOT={GUN[] "3                       ",RETR_CMD[] "#OPN                    ",CHOISE[] "#FIRST                  ",CLO_TM[] "1                       ",PGNO1[] "197                     ",PRESS1[] "0                       ",PGNO2[] "1                       ",PRESS2[] "0                       ",SPOT_PARAMS[] "NORMAL                  "}
DECL BASIS_SUGG_T LAST_BASIS={POINT1[] "SWP_60_9234             ",POINT2[] "SWP_60_9234             ",CP_PARAMS[] "CPDAT30                 ",PTP_PARAMS[] "PDAT38                  ",CONT[] "                        ",CP_VEL[] "2                       ",PTP_VEL[] "100                     "}
DECL E6POS XSWP_60_7258={x 177.344299,y 91.2774734,z 492.510498,a -80.9878082,b 30.2983799,c 107.447899,s 2,t 11,e1 0.0,e2 0.0,e3 0.0,e4 0.0,e5 0.0,e6 0.0}
DECL FDAT FSWP_60_7258={TOOL_NO 3,BASE_NO 3,IPO_FRAME #BASE}
DECL E6POS XSWP_60_7217={x 212.0215,y -5.72816896,z 386.457611,a -89.9976273,b 44.4766617,c 89.9928436,s 2,t 43,e1 0.0,e2 0.0,e3 0.0,e4 0.0,e5 0.0,e6 0.0}
DECL FDAT FSWP_60_7217={TOOL_NO 3,BASE_NO 3,IPO_FRAME #BASE}
DECL E6POS XSWP_60_7218={x 230.446198,y 232.953796,z 499.446594,a -89.995369,b 44.4764595,c 89.9949036,s 2,t 43,e1 0.0,e2 0.0,e3 0.0,e4 0.0,e5 0.0,e6 0.0}
DECL FDAT FSWP_60_7218={TOOL_NO 3,BASE_NO 3,IPO_FRAME #BASE}
DECL PDAT PPDAT1={VEL 100.0,ACC 100.0,APO_DIST 0.0}
DECL E6POS XSWP_60_7253={x 183.271103,y -168.511398,z 488.607788,a -80.492569,b 31.5890808,c 107.705902,s 2,t 43,e1 0.0,e2 0.0,e3 0.0,e4 0.0,e5 0.0,e6 0.0}
DECL FDAT FSWP_60_7253={TOOL_NO 3,BASE_NO 3,IPO_FRAME #BASE}
DECL E6POS XSWP_60_7255={x 182.816605,y -136.932495,z 488.353302,a -80.4999466,b 31.6015491,c 107.701401,s 2,t 43,e1 0.0,e2 0.0,e3 0.0,e4 0.0,e5 0.0,e6 0.0}
DECL FDAT FSWP_60_7255={TOOL_NO 3,BASE_NO 3,IPO_FRAME #BASE}
DECL E6POS XSWP_60_7257={x 182.301605,y -88.3556519,z 488.131897,a -80.5033569,b 31.6069908,c 107.6978,s 2,t 43,e1 0.0,e2 0.0,e3 0.0,e4 0.0,e5 0.0,e6 0.0}
DECL FDAT FSWP_60_7257={TOOL_NO 3,BASE_NO 3,IPO_FRAME #BASE}
DECL E6POS XSWP_60_7262={x 180.669205,y 1.25821102,z 490.930298,a -80.508873,b 31.6130199,c 107.696198,s 2,t 11,e1 0.0,e2 0.0,e3 0.0,e4 0.0,e5 0.0,e6 0.0}
DECL FDAT FSWP_60_7262={TOOL_NO 3,BASE_NO 3,IPO_FRAME #BASE}
DECL SPOT_TYPE SNORMAL
DECL SPOT_TYPE SNORMAL28
DECL E6POS XP15={x -800.207581,y 1052.86096,z 371.426514,a 42.3493195,b -1.00002205,c -26.3774109,s 2,t 42,e1 0.0,e2 0.0,e3 0.0,e4 0.0,e5 0.0,e6 0.0}
DECL FDAT FP15={TOOL_NO 1,BASE_NO 3,IPO_FRAME #BASE}
DECL PDAT PPDAT2={VEL 100.0,ACC 100.0,APO_DIST 100.0}
DECL E6POS Xl048={x 235.096298,y 205.879898,z 399.392609,a -89.9929504,b 44.4753685,c 89.9981766,s 2,t 43,e1 0.0,e2 0.0,e3 0.0,e4 0.0,e5 0.0,e6 0.0}
DECL FDAT Fl048={TOOL_NO 3,BASE_NO 3,IPO_FRAME #BASE}
DECL PDAT PP_OLP53={VEL 100.0,ACC 100.0,APO_DIST 0.0}
DECL LDAT LL_OLP50={VEL 2.0,ACC 100.0,APO_DIST 0.0,APO_FAC 0.0}
DECL SPOT_TYPE SNORMAL29
DECL LDAT LCPDAT5={VEL 2.0,ACC 100.0,APO_DIST 100.0,APO_FAC 50.0}
DECL LDAT LCPDAT6={VEL 2.0,ACC 100.0,APO_DIST 100.0,APO_FAC 50.0}
DECL E6POS XP16={x 208.831604,y -34.5271187,z 495.562012,a -80.5012817,b 31.5980301,c 107.702202,s 2,t 11,e1 0.0,e2 0.0,e3 0.0,e4 0.0,e5 0.0,e6 0.0}
DECL FDAT FP16={TOOL_NO 3,BASE_NO 3,IPO_FRAME #BASE}
DECL LDAT LCPDAT7={VEL 2.0,ACC 50.0,APO_DIST 100.0,APO_FAC 50.0}
DECL E6POS XSWP_60_7381={x 206.840393,y 416.639099,z 400.304108,a -89.9998703,b 62.6937904,c 90.0006027,s 2,t 43,e1 0.0,e2 0.0,e3 0.0,e4 0.0,e5 0.0,e6 0.0}
DECL FDAT FSWP_60_7381={TOOL_NO 3,BASE_NO 3,IPO_FRAME #BASE}
DECL LDAT LL_OLP16={VEL 2.0,ACC 100.0,APO_DIST 0.0,APO_FAC 0.0}
DECL SPOT_TYPE SNORMAL13
DECL E6POS XSWP_60_7382={x 206.840393,y 416.639099,z 400.304108,a -89.9998703,b 62.6937904,c 90.0006027,s 2,t 43,e1 0.0,e2 0.0,e3 0.0,e4 0.0,e5 0.0,e6 0.0}
DECL FDAT FSWP_60_7382={TOOL_NO 3,BASE_NO 3,IPO_FRAME #BASE}
DECL LDAT LL_OLP17={VEL 2.0,ACC 100.0,APO_DIST 0.0,APO_FAC 0.0}
DECL E6POS XSWP_60_7383={x 206.840393,y 416.639099,z 400.304108,a -89.9998703,b 62.6937904,c 90.0006027,s 2,t 43,e1 0.0,e2 0.0,e3 0.0,e4 0.0,e5 0.0,e6 0.0}
DECL FDAT FSWP_60_7383={TOOL_NO 3,BASE_NO 3,IPO_FRAME #BASE}
DECL LDAT LL_OLP18={VEL 2.0,ACC 100.0,APO_DIST 0.0,APO_FAC 0.0}
DECL E6POS XSWP_60_7384={x 206.840393,y 416.639099,z 400.304108,a -89.9998703,b 62.6937904,c 90.0006027,s 2,t 43,e1 0.0,e2 0.0,e3 0.0,e4 0.0,e5 0.0,e6 0.0}
DECL FDAT FSWP_60_7384={TOOL_NO 3,BASE_NO 3,IPO_FRAME #BASE}
DECL LDAT LL_OLP19={VEL 2.0,ACC 100.0,APO_DIST 0.0,APO_FAC 0.0}
DECL E6POS XSWP_60_7385={x 206.840393,y 416.639099,z 400.304108,a -89.9998703,b 62.6937904,c 90.0006027,s 2,t 43,e1 0.0,e2 0.0,e3 0.0,e4 0.0,e5 0.0,e6 0.0}
DECL FDAT FSWP_60_7385={TOOL_NO 3,BASE_NO 3,IPO_FRAME #BASE}
DECL LDAT LL_OLP20={VEL 2.0,ACC 100.0,APO_DIST 0.0,APO_FAC 0.0}
DECL E6POS XP17={x 487.528015,y 470.183289,z 402.488708,a 89.9994965,b -2.90493488,c -90.0005722,s 2,t 43,e1 0.0,e2 0.0,e3 0.0,e4 0.0,e5 0.0,e6 0.0}
DECL FDAT FP17={TOOL_NO 1,BASE_NO 3,IPO_FRAME #BASE}
DECL PDAT PPDAT5={VEL 100.0,ACC 80.0,APO_DIST 100.0}
DECL E6POS XSWP_60_9230={x 211.793198,y 368.260498,z 385.74881,a -89.9941635,b 62.6974602,c 90.0023727,s 2,t 43,e1 0.0,e2 0.0,e3 0.0,e4 0.0,e5 0.0,e6 0.0}
DECL FDAT FSWP_60_9230={TOOL_NO 3,BASE_NO 3,IPO_FRAME #BASE}
DECL E6POS XSWP_60_7230={x 206.551697,y 281.323212,z 384.273712,a -89.9992828,b 62.6938591,c 90.0016403,s 2,t 43,e1 0.0,e2 0.0,e3 0.0,e4 0.0,e5 0.0,e6 0.0}
DECL FDAT FSWP_60_7230={TOOL_NO 3,BASE_NO 3,IPO_FRAME #BASE}
DECL E6POS XSWP_60_9224={x 212.402298,y 237.695206,z 382.723602,a -90.0041122,b 62.6942406,c 89.9951477,s 2,t 43,e1 0.0,e2 0.0,e3 0.0,e4 0.0,e5 0.0,e6 0.0}
DECL FDAT FSWP_60_9224={TOOL_NO 3,BASE_NO 3,IPO_FRAME #BASE}
DECL E6POS XSWP_60_9222={x 213.050293,y 187.744598,z 382.238586,a -90.0049973,b 62.6928902,c 89.9948196,s 2,t 43,e1 0.0,e2 0.0,e3 0.0,e4 0.0,e5 0.0,e6 0.0}
DECL FDAT FSWP_60_9222={TOOL_NO 3,BASE_NO 3,IPO_FRAME #BASE}
DECL E6POS XSWP_60_9220={x 213.400696,y 141.378403,z 382.481903,a -90.0000381,b 54.2503891,c 89.9955215,s 2,t 43,e1 0.0,e2 0.0,e3 0.0,e4 0.0,e5 0.0,e6 0.0}
DECL FDAT FSWP_60_9220={TOOL_NO 3,BASE_NO 3,IPO_FRAME #BASE}
DECL E6POS XP18={x 479.408508,y 208.821899,z 388.631012,a 90.0012131,b -2.90534997,c -90.0033875,s 2,t 43,e1 0.0,e2 0.0,e3 0.0,e4 0.0,e5 0.0,e6 0.0}
DECL FDAT FP18={TOOL_NO 1,BASE_NO 3,IPO_FRAME #BASE}
DECL PDAT PPDAT8={VEL 100.0,ACC 80.0,APO_DIST 100.0}
DECL E6POS XSWP_60_7223={x 211.064697,y 88.1381378,z 386.404205,a -89.9957275,b 44.4758797,c 89.9949112,s 2,t 43,e1 0.0,e2 0.0,e3 0.0,e4 0.0,e5 0.0,e6 0.0}
DECL FDAT FSWP_60_7223={TOOL_NO 3,BASE_NO 3,IPO_FRAME #BASE}
DECL LDAT LCPDAT8={VEL 2.0,ACC 100.0,APO_DIST 100.0,APO_FAC 50.0}
DECL SPOT_TYPE SNORMAL1
DECL E6POS XSWP_60_7219={x 212.021896,y -5.72421885,z 386.506012,a -89.9952469,b 44.4766808,c 89.9958267,s 2,t 43,e1 0.0,e2 0.0,e3 0.0,e4 0.0,e5 0.0,e6 0.0}
DECL FDAT FSWP_60_7219={TOOL_NO 3,BASE_NO 3,IPO_FRAME #BASE}
DECL LDAT LL_OLP51={VEL 2.0,ACC 100.0,APO_DIST 0.0,APO_FAC 0.0}
DECL E6POS XP19={x 456.774689,y 152.085098,z 534.078979,a 82.0662766,b 27.2542496,c -106.930702,s 2,t 11,e1 0.0,e2 0.0,e3 0.0,e4 0.0,e5 0.0,e6 0.0}
DECL FDAT FP19={TOOL_NO 1,BASE_NO 3,IPO_FRAME #BASE}
DECL PDAT PPDAT9={VEL 100.0,ACC 80.0,APO_DIST 100.0}
DECL E6POS XP20={x 463.799011,y 181.4142,z 472.935089,a 88.6661911,b 4.65849304,c -105.848,s 2,t 43,e1 0.0,e2 0.0,e3 0.0,e4 0.0,e5 0.0,e6 0.0}
DECL FDAT FP20={TOOL_NO 1,BASE_NO 3,IPO_FRAME #BASE}
DECL PDAT PPDAT10={VEL 100.0,ACC 80.0,APO_DIST 100.0}
DECL E6POS XSWP_60_7259={x 186.947998,y 91.3792191,z 492.51651,a -80.987381,b 30.2990799,c 107.448097,s 2,t 11,e1 0.0,e2 0.0,e3 0.0,e4 0.0,e5 0.0,e6 0.0}
DECL FDAT FSWP_60_7259={TOOL_NO 3,BASE_NO 3,IPO_FRAME #BASE}
DECL LDAT LL_OLP39={VEL 2.0,ACC 100.0,APO_DIST 0.0,APO_FAC 0.0}
DECL SPOT_TYPE SNORMAL36
DECL E6POS XSWP_60_7263={x 186.947998,y 91.3792191,z 492.51651,a -80.987381,b 30.2990799,c 107.448097,s 2,t 11,e1 0.0,e2 0.0,e3 0.0,e4 0.0,e5 0.0,e6 0.0}
DECL FDAT FSWP_60_7263={TOOL_NO 3,BASE_NO 3,IPO_FRAME #BASE}
DECL LDAT LL_OLP40={VEL 2.0,ACC 100.0,APO_DIST 0.0,APO_FAC 0.0}
DECL E6POS XSWP_60_7264={x 186.947998,y 91.3792191,z 492.51651,a -80.987381,b 30.2990799,c 107.448097,s 2,t 11,e1 0.0,e2 0.0,e3 0.0,e4 0.0,e5 0.0,e6 0.0}
DECL FDAT FSWP_60_7264={TOOL_NO 3,BASE_NO 3,IPO_FRAME #BASE}
DECL LDAT LL_OLP41={VEL 2.0,ACC 100.0,APO_DIST 0.0,APO_FAC 0.0}
DECL E6POS XSWP_60_7265={x 186.947998,y 91.3792191,z 492.51651,a -80.987381,b 30.2990799,c 107.448097,s 2,t 11,e1 0.0,e2 0.0,e3 0.0,e4 0.0,e5 0.0,e6 0.0}
DECL FDAT FSWP_60_7265={TOOL_NO 3,BASE_NO 3,IPO_FRAME #BASE}
DECL LDAT LL_OLP42={VEL 2.0,ACC 100.0,APO_DIST 0.0,APO_FAC 0.0}
DECL E6POS XSWP_60_7266={x 186.947998,y 91.3792191,z 492.51651,a -80.987381,b 30.2990799,c 107.448097,s 2,t 11,e1 0.0,e2 0.0,e3 0.0,e4 0.0,e5 0.0,e6 0.0}
DECL FDAT FSWP_60_7266={TOOL_NO 3,BASE_NO 3,IPO_FRAME #BASE}
DECL LDAT LL_OLP43={VEL 2.0,ACC 100.0,APO_DIST 0.0,APO_FAC 0.0}
DECL E6POS XSWP_60_7267={x 186.947998,y 91.3792191,z 492.51651,a -80.987381,b 30.2990799,c 107.448097,s 2,t 11,e1 0.0,e2 0.0,e3 0.0,e4 0.0,e5 0.0,e6 0.0}
DECL FDAT FSWP_60_7267={TOOL_NO 3,BASE_NO 3,IPO_FRAME #BASE}
DECL LDAT LL_OLP44={VEL 2.0,ACC 100.0,APO_DIST 0.0,APO_FAC 0.0}
DECL E6POS XSWP_60_7268={x 186.947998,y 91.3792191,z 492.51651,a -80.987381,b 30.2990799,c 107.448097,s 2,t 11,e1 0.0,e2 0.0,e3 0.0,e4 0.0,e5 0.0,e6 0.0}
DECL FDAT FSWP_60_7268={TOOL_NO 3,BASE_NO 3,IPO_FRAME #BASE}
DECL LDAT LL_OLP45={VEL 2.0,ACC 100.0,APO_DIST 0.0,APO_FAC 0.0}
DECL E6POS XSWP_60_7269={x 186.947998,y 91.3792191,z 492.51651,a -80.987381,b 30.2990799,c 107.448097,s 2,t 11,e1 0.0,e2 0.0,e3 0.0,e4 0.0,e5 0.0,e6 0.0}
DECL FDAT FSWP_60_7269={TOOL_NO 3,BASE_NO 3,IPO_FRAME #BASE}
DECL LDAT LL_OLP46={VEL 2.0,ACC 100.0,APO_DIST 0.0,APO_FAC 0.0}
DECL E6POS XSWP_60_7270={x 186.947998,y 91.3792191,z 492.51651,a -80.987381,b 30.2990799,c 107.448097,s 2,t 11,e1 0.0,e2 0.0,e3 0.0,e4 0.0,e5 0.0,e6 0.0}
DECL FDAT FSWP_60_7270={TOOL_NO 3,BASE_NO 3,IPO_FRAME #BASE}
DECL LDAT LL_OLP47={VEL 2.0,ACC 100.0,APO_DIST 0.0,APO_FAC 0.0}
DECL E6POS XSWP_60_7271={x 186.947998,y 91.3792191,z 492.51651,a -80.987381,b 30.2990799,c 107.448097,s 2,t 11,e1 0.0,e2 0.0,e3 0.0,e4 0.0,e5 0.0,e6 0.0}
DECL FDAT FSWP_60_7271={TOOL_NO 3,BASE_NO 3,IPO_FRAME #BASE}
DECL LDAT LL_OLP48={VEL 2.0,ACC 100.0,APO_DIST 0.0,APO_FAC 0.0}
DECL E6POS XSWP_60_7272={x 186.947998,y 91.3792191,z 492.51651,a -80.987381,b 30.2990799,c 107.448097,s 2,t 11,e1 0.0,e2 0.0,e3 0.0,e4 0.0,e5 0.0,e6 0.0}
DECL FDAT FSWP_60_7272={TOOL_NO 3,BASE_NO 3,IPO_FRAME #BASE}
DECL LDAT LL_OLP49={VEL 2.0,ACC 100.0,APO_DIST 0.0,APO_FAC 0.0}
DECL E6POS XSWP_60_7273={x 186.947998,y 91.3792191,z 492.51651,a -80.987381,b 30.2990799,c 107.448097,s 2,t 11,e1 0.0,e2 0.0,e3 0.0,e4 0.0,e5 0.0,e6 0.0}
DECL FDAT FSWP_60_7273={TOOL_NO 3,BASE_NO 3,IPO_FRAME #BASE}
DECL LDAT LL_OLP52={VEL 2.0,ACC 100.0,APO_DIST 0.0,APO_FAC 0.0}
DECL E6POS XSWP_60_9308={x 206.887207,y 113.207497,z 405.258209,a -73.527977,b 45.4203415,c 112.484299,s 2,t 43,e1 0.0,e2 0.0,e3 0.0,e4 0.0,e5 0.0,e6 0.0}
DECL FDAT FSWP_60_9308={TOOL_NO 3,BASE_NO 3,IPO_FRAME #BASE}
DECL E6POS XSWP_60_9310={x 201.055801,y 113.228104,z 431.161285,a -73.5282288,b 45.4178314,c 112.4842,s 2,t 43,e1 0.0,e2 0.0,e3 0.0,e4 0.0,e5 0.0,e6 0.0}
DECL FDAT FSWP_60_9310={TOOL_NO 3,BASE_NO 3,IPO_FRAME #BASE}
DECL E6POS XSWP_60_9212={x 193.817001,y 112.206703,z 460.553802,a -73.5267792,b 45.4153099,c 112.485397,s 2,t 43,e1 0.0,e2 0.0,e3 0.0,e4 0.0,e5 0.0,e6 0.0}
DECL FDAT FSWP_60_9212={TOOL_NO 3,BASE_NO 3,IPO_FRAME #BASE}
DECL E6POS XSWP_60_9250={x 184.402405,y 131.005402,z 489.79541,a -73.5274582,b 45.41576,c 112.485397,s 2,t 43,e1 0.0,e2 0.0,e3 0.0,e4 0.0,e5 0.0,e6 0.0}
DECL FDAT FSWP_60_9250={TOOL_NO 3,BASE_NO 3,IPO_FRAME #BASE}
DECL E6POS XSWP_60_9248={x 184.599106,y 168.533707,z 489.699188,a -73.527153,b 45.4180298,c 112.485199,s 2,t 43,e1 0.0,e2 0.0,e3 0.0,e4 0.0,e5 0.0,e6 0.0}
DECL FDAT FSWP_60_9248={TOOL_NO 3,BASE_NO 3,IPO_FRAME #BASE}
DECL E6POS XSWP_60_9246={x 183.884506,y 206.977905,z 489.657898,a -73.5289536,b 45.4170799,c 112.4841,s 2,t 11,e1 0.0,e2 0.0,e3 0.0,e4 0.0,e5 0.0,e6 0.0}
DECL FDAT FSWP_60_9246={TOOL_NO 3,BASE_NO 3,IPO_FRAME #BASE}
DECL E6POS XSWP_60_9244={x 184.423203,y 249.814804,z 489.650391,a -73.5230331,b 45.4163399,c 112.489502,s 2,t 11,e1 0.0,e2 0.0,e3 0.0,e4 0.0,e5 0.0,e6 0.0}
DECL FDAT FSWP_60_9244={TOOL_NO 3,BASE_NO 3,IPO_FRAME #BASE}
DECL E6POS XSWP_60_9242={x 185.195007,y 285.5513,z 487.9776,a -73.5297318,b 45.4183388,c 112.4842,s 2,t 11,e1 0.0,e2 0.0,e3 0.0,e4 0.0,e5 0.0,e6 0.0}
DECL FDAT FSWP_60_9242={TOOL_NO 3,BASE_NO 3,IPO_FRAME #BASE}
DECL E6POS XSWP_60_9240={x 183.838699,y 324.021515,z 488.159088,a -73.5266724,b 45.4191017,c 112.485397,s 2,t 11,e1 0.0,e2 0.0,e3 0.0,e4 0.0,e5 0.0,e6 0.0}
DECL FDAT FSWP_60_9240={TOOL_NO 3,BASE_NO 3,IPO_FRAME #BASE}
DECL E6POS XSWP_60_9238={x 184.964203,y 365.820801,z 487.026611,a -73.5268936,b 45.4204216,c 112.485298,s 2,t 11,e1 0.0,e2 0.0,e3 0.0,e4 0.0,e5 0.0,e6 0.0}
DECL FDAT FSWP_60_9238={TOOL_NO 3,BASE_NO 3,IPO_FRAME #BASE}
DECL E6POS XSWP_60_9236={x 191.128906,y 385.006104,z 461.481506,a -43.1879387,b 69.0690994,c 138.713104,s 2,t 43,e1 0.0,e2 0.0,e3 0.0,e4 0.0,e5 0.0,e6 0.0}
DECL FDAT FSWP_60_9236={TOOL_NO 3,BASE_NO 3,IPO_FRAME #BASE}
DECL E6POS XSWP_60_9232={x 212.561005,y 281.382294,z 383.535614,a -90.0006485,b 62.6943016,c 90.000061,s 2,t 43,e1 0.0,e2 0.0,e3 0.0,e4 0.0,e5 0.0,e6 0.0}
DECL FDAT FSWP_60_9232={TOOL_NO 3,BASE_NO 3,IPO_FRAME #BASE}
DECL E6POS XP21={x 433.752899,y 464.826813,z 652.343994,a 88.1901703,b 6.72100019,c -105.1064,s 2,t 11,e1 0.0,e2 0.0,e3 0.0,e4 0.0,e5 0.0,e6 0.0}
DECL FDAT FP21={TOOL_NO 1,BASE_NO 3,IPO_FRAME #BASE}
DECL PDAT PPDAT11={VEL 100.0,ACC 80.0,APO_DIST 100.0}
DECL E6POS XP22={x 440.558899,y 443.846893,z 605.240601,a 89.9558334,b -0.390211314,c -102.807098,s 2,t 43,e1 0.0,e2 0.0,e3 0.0,e4 0.0,e5 0.0,e6 0.0}
DECL FDAT FP22={TOOL_NO 1,BASE_NO 3,IPO_FRAME #BASE}
DECL PDAT PPDAT12={VEL 100.0,ACC 80.0,APO_DIST 100.0}
DECL E6POS XP23={x 467.926392,y 448.115997,z 544.223999,a 94.4578781,b -15.4472399,c -106.169296,s 2,t 43,e1 0.0,e2 0.0,e3 0.0,e4 0.0,e5 0.0,e6 0.0}
DECL FDAT FP23={TOOL_NO 1,BASE_NO 3,IPO_FRAME #BASE}
DECL PDAT PPDAT13={VEL 100.0,ACC 80.0,APO_DIST 100.0}
DECL PDAT PPDAT14={VEL 100.0,ACC 80.0,APO_DIST 100.0}
DECL LDAT LCPDAT9={VEL 2.0,ACC 100.0,APO_DIST 100.0,APO_FAC 50.0}
DECL PDAT PPDAT15={VEL 100.0,ACC 80.0,APO_DIST 100.0}
DECL LDAT LCPDAT10={VEL 2.0,ACC 100.0,APO_DIST 100.0,APO_FAC 50.0}
DECL E6POS XP12={x 468.767487,y -1397.66797,z 1152.35498,a 140.2052,b 16.2280006,c 9.75706577,s 2,t 34,e1 0.0,e2 0.0,e3 0.0,e4 0.0,e5 0.0,e6 0.0}
DECL FDAT FP12={TOOL_NO 3,BASE_NO 0,IPO_FRAME #BASE}
DECL PDAT PPDAT16={VEL 100.0,ACC 80.0,APO_DIST 100.0}
DECL E6POS XP13={x 468.767487,y -1397.66797,z 1152.35498,a 140.2052,b 16.2280006,c 9.75706577,s 2,t 34,e1 0.0,e2 0.0,e3 0.0,e4 0.0,e5 0.0,e6 0.0}
DECL FDAT FP13={TOOL_NO 3,BASE_NO 0,IPO_FRAME #BASE}
DECL PDAT PPDAT17={VEL 100.0,ACC 80.0,APO_DIST 100.0}
DECL E6POS XP14={x 468.767487,y -1397.66797,z 1152.35498,a 140.2052,b 16.2280006,c 9.75706577,s 2,t 34,e1 0.0,e2 0.0,e3 0.0,e4 0.0,e5 0.0,e6 0.0}
DECL FDAT FP14={TOOL_NO 3,BASE_NO 0,IPO_FRAME #BASE}
DECL PDAT PPDAT18={VEL 100.0,ACC 80.0,APO_DIST 100.0}
DECL E6POS XP24={x 468.767487,y -1397.66797,z 1152.35498,a 140.2052,b 16.2280006,c 9.75706577,s 2,t 34,e1 0.0,e2 0.0,e3 0.0,e4 0.0,e5 0.0,e6 0.0}
DECL FDAT FP24={TOOL_NO 3,BASE_NO 0,IPO_FRAME #BASE}
DECL PDAT PPDAT19={VEL 100.0,ACC 80.0,APO_DIST 100.0}
DECL E6POS XP25={x -384.03299,y 419.546387,z 316.5065,a 66.1975403,b -17.4831791,c -68.3892136,s 2,t 42,e1 0.0,e2 0.0,e3 0.0,e4 0.0,e5 0.0,e6 0.0}
DECL FDAT FP25={TOOL_NO 3,BASE_NO 3,IPO_FRAME #BASE}
DECL PDAT PPDAT20={VEL 100.0,ACC 80.0,APO_DIST 100.0}
DECL E6POS XP26={x 202.700699,y 221.683807,z 190.377502,a 83.5018692,b -22.9824409,c -74.4219131,s 2,t 43,e1 0.0,e2 0.0,e3 0.0,e4 0.0,e5 0.0,e6 0.0}
DECL FDAT FP26={TOOL_NO 3,BASE_NO 3,IPO_FRAME #BASE}
DECL PDAT PPDAT21={VEL 100.0,ACC 80.0,APO_DIST 100.0}
DECL E6POS XP27={x 187.651306,y 27.2828407,z 289.910187,a 88.4408417,b -40.7095108,c -87.5350037,s 2,t 43,e1 0.0,e2 0.0,e3 0.0,e4 0.0,e5 0.0,e6 0.0}
DECL FDAT FP27={TOOL_NO 3,BASE_NO 3,IPO_FRAME #BASE}
DECL LDAT LCPDAT11={VEL 2.0,ACC 100.0,APO_DIST 100.0,APO_FAC 50.0}
DECL E6POS XP28={x 186.2314,y 169.758194,z 261.008087,a 88.6298065,b -33.4667816,c -87.8612366,s 2,t 43,e1 0.0,e2 0.0,e3 0.0,e4 0.0,e5 0.0,e6 0.0}
DECL FDAT FP28={TOOL_NO 3,BASE_NO 3,IPO_FRAME #BASE}
DECL PDAT PPDAT22={VEL 100.0,ACC 80.0,APO_DIST 100.0}
DECL E6POS XSWP_60_7160={x 187.652405,y 27.2816505,z 289.94101,a 88.4419098,b -40.7085609,c -87.5364304,s 2,t 43,e1 0.0,e2 0.0,e3 0.0,e4 0.0,e5 0.0,e6 0.0}
DECL FDAT FSWP_60_7160={TOOL_NO 3,BASE_NO 3,IPO_FRAME #BASE}
DECL E6POS XP29={x 187.294296,y 62.0672302,z 289.905487,a 88.4418106,b -40.7092781,c -87.536438,s 2,t 43,e1 0.0,e2 0.0,e3 0.0,e4 0.0,e5 0.0,e6 0.0}
DECL FDAT FP29={TOOL_NO 3,BASE_NO 3,IPO_FRAME #BASE}
DECL LDAT LCPDAT12={VEL 2.0,ACC 100.0,APO_DIST 100.0,APO_FAC 50.0}
DECL E6POS XP30={x 186.636307,y 125.065102,z 289.793213,a 88.440773,b -40.712059,c -87.5349197,s 2,t 43,e1 0.0,e2 0.0,e3 0.0,e4 0.0,e5 0.0,e6 0.0}
DECL FDAT FP30={TOOL_NO 3,BASE_NO 3,IPO_FRAME #BASE}
DECL LDAT LCPDAT13={VEL 2.0,ACC 100.0,APO_DIST 100.0,APO_FAC 50.0}
DECL E6POS XSWP_60_7158={x 187.294296,y 62.0672302,z 289.905487,a 88.4418106,b -40.7092781,c -87.536438,s 2,t 43,e1 0.0,e2 0.0,e3 0.0,e4 0.0,e5 0.0,e6 0.0}
DECL FDAT FSWP_60_7158={TOOL_NO 3,BASE_NO 3,IPO_FRAME #BASE}
DECL E6POS XSWP_60_7154={x 186.636307,y 125.065102,z 289.793213,a 88.440773,b -40.712059,c -87.5349197,s 2,t 43,e1 0.0,e2 0.0,e3 0.0,e4 0.0,e5 0.0,e6 0.0}
DECL FDAT FSWP_60_7154={TOOL_NO 3,BASE_NO 3,IPO_FRAME #BASE}
DECL E6POS XSWP_60_7152={x 186.402603,y 149.349899,z 289.780396,a 88.4422379,b -40.7125282,c -87.5355225,s 2,t 43,e1 0.0,e2 0.0,e3 0.0,e4 0.0,e5 0.0,e6 0.0}
DECL FDAT FSWP_60_7152={TOOL_NO 3,BASE_NO 3,IPO_FRAME #BASE}
DECL LDAT LCPDAT14={VEL 2.0,ACC 100.0,APO_DIST 100.0,APO_FAC 50.0}
DECL E6POS XSWP_60_7150={x 184.194901,y 177.324402,z 291.644012,a 88.4415131,b -40.7133217,c -87.5351028,s 2,t 43,e1 0.0,e2 0.0,e3 0.0,e4 0.0,e5 0.0,e6 0.0}
DECL FDAT FSWP_60_7150={TOOL_NO 3,BASE_NO 3,IPO_FRAME #BASE}
DECL LDAT LCPDAT15={VEL 2.0,ACC 100.0,APO_DIST 100.0,APO_FAC 50.0}
DECL E6POS XSWP_60_7148={x 183.885406,y 206.6828,z 291.57309,a 88.4399872,b -40.71521,c -87.5329819,s 2,t 43,e1 0.0,e2 0.0,e3 0.0,e4 0.0,e5 0.0,e6 0.0}
DECL FDAT FSWP_60_7148={TOOL_NO 3,BASE_NO 3,IPO_FRAME #BASE}
DECL LDAT LCPDAT16={VEL 2.0,ACC 100.0,APO_DIST 100.0,APO_FAC 50.0}
DECL E6POS XSWP_60_7146={x 183.580994,y 235.289093,z 291.526611,a 88.4393768,b -40.7172585,c -87.5320663,s 2,t 43,e1 0.0,e2 0.0,e3 0.0,e4 0.0,e5 0.0,e6 0.0}
DECL FDAT FSWP_60_7146={TOOL_NO 3,BASE_NO 3,IPO_FRAME #BASE}
DECL LDAT LCPDAT17={VEL 2.0,ACC 100.0,APO_DIST 100.0,APO_FAC 50.0}
DECL E6POS XSWP_60_7144={x 183.271698,y 265.554901,z 291.498596,a 88.4393463,b -40.7176704,c -87.5321884,s 2,t 43,e1 0.0,e2 0.0,e3 0.0,e4 0.0,e5 0.0,e6 0.0}
DECL FDAT FSWP_60_7144={TOOL_NO 3,BASE_NO 3,IPO_FRAME #BASE}
DECL LDAT LCPDAT18={VEL 2.0,ACC 100.0,APO_DIST 100.0,APO_FAC 50.0}
DECL E6POS XSWP_60_7142={x 182.987595,y 294.084503,z 291.476715,a 88.4403076,b -40.719059,c -87.5332031,s 2,t 43,e1 0.0,e2 0.0,e3 0.0,e4 0.0,e5 0.0,e6 0.0}
DECL FDAT FSWP_60_7142={TOOL_NO 3,BASE_NO 3,IPO_FRAME #BASE}
DECL LDAT LCPDAT19={VEL 2.0,ACC 100.0,APO_DIST 100.0,APO_FAC 50.0}
DECL E6POS XSWP_60_7140={x 182.677307,y 324.696899,z 291.416504,a 88.4400635,b -40.7207718,c -87.5320663,s 2,t 43,e1 0.0,e2 0.0,e3 0.0,e4 0.0,e5 0.0,e6 0.0}
DECL FDAT FSWP_60_7140={TOOL_NO 3,BASE_NO 3,IPO_FRAME #BASE}
DECL LDAT LCPDAT20={VEL 2.0,ACC 100.0,APO_DIST 100.0,APO_FAC 50.0}
DECL E6POS XSWP_60_7136={x 183.638,y 354.853912,z 283.04599,a 88.4401169,b -40.7217407,c -87.5323563,s 2,t 43,e1 0.0,e2 0.0,e3 0.0,e4 0.0,e5 0.0,e6 0.0}
DECL FDAT FSWP_60_7136={TOOL_NO 3,BASE_NO 3,IPO_FRAME #BASE}
DECL LDAT LCPDAT21={VEL 2.0,ACC 100.0,APO_DIST 100.0,APO_FAC 50.0}
DECL E6POS XSWP_60_7137={x 188.785202,y 354.862701,z 240.309402,a 88.4393768,b -40.723999,c -87.5315781,s 2,t 43,e1 0.0,e2 0.0,e3 0.0,e4 0.0,e5 0.0,e6 0.0}
DECL FDAT FSWP_60_7137={TOOL_NO 3,BASE_NO 3,IPO_FRAME #BASE}
DECL PDAT PPDAT23={VEL 100.0,ACC 80.0,APO_DIST 100.0}
DECL E6POS XPS_30={x 8.17374325,y 352.267487,z 239.812698,a 88.4372711,b -40.7192917,c -87.5370407,s 2,t 43,e1 0.0,e2 0.0,e3 0.0,e4 0.0,e5 0.0,e6 0.0}
DECL FDAT FPS_30={TOOL_NO 3,BASE_NO 3,IPO_FRAME #BASE}
DECL PDAT PPDAT24={VEL 100.0,ACC 80.0,APO_DIST 100.0}
DECL E6POS XPS_31={x 8.17374325,y 352.267487,z 239.812698,a 88.4372711,b -40.7192917,c -87.5370407,s 2,t 43,e1 0.0,e2 0.0,e3 0.0,e4 0.0,e5 0.0,e6 0.0}
DECL FDAT FPS_31={TOOL_NO 3,BASE_NO 3,IPO_FRAME #BASE}
DECL PDAT PPDAT25={VEL 100.0,ACC 80.0,APO_DIST 100.0}
DECL E6POS XPS_32={x -352.048706,y 791.363525,z 674.182678,a 102.5298,b 65.7294617,c -50.9808998,s 2,t 42,e1 0.0,e2 0.0,e3 0.0,e4 0.0,e5 0.0,e6 0.0}
DECL FDAT FPS_32={TOOL_NO 3,BASE_NO 3,IPO_FRAME #BASE}
DECL PDAT PPDAT26={VEL 100.0,ACC 80.0,APO_DIST 100.0}
DECL E6POS XPS_33={x 187.030197,y 354.844299,z 237.620605,a 88.438652,b -40.7234612,c -87.5300064,s 2,t 43,e1 0.0,e2 0.0,e3 0.0,e4 0.0,e5 0.0,e6 0.0}
DECL FDAT FPS_33={TOOL_NO 3,BASE_NO 3,IPO_FRAME #BASE}
DECL PDAT PPDAT27={VEL 100.0,ACC 80.0,APO_DIST 100.0}
DECL E6POS XPS_34={x -938.618225,y 703.747803,z 612.635803,a 165.016998,b 23.1207695,c 13.1032801,s 2,t 42,e1 0.0,e2 0.0,e3 0.0,e4 0.0,e5 0.0,e6 0.0}
DECL FDAT FPS_34={TOOL_NO 3,BASE_NO 3,IPO_FRAME #BASE}
DECL PDAT PPDAT28={VEL 100.0,ACC 80.0,APO_DIST 100.0}
DECL E6POS XPS_35={x -373.168396,y 990.912476,z -71.8266068,a 96.466713,b 6.40488195,c -88.1943283,s 2,t 42,e1 0.0,e2 0.0,e3 0.0,e4 0.0,e5 0.0,e6 0.0}
DECL FDAT FPS_35={TOOL_NO 3,BASE_NO 3,IPO_FRAME #BASE}
DECL PDAT PPDAT29={VEL 100.0,ACC 80.0,APO_DIST 100.0}
DECL E6POS XPS_36={x -367.697113,y 444.486786,z -71.2692413,a 96.4659195,b 6.40667391,c -88.1916122,s 2,t 42,e1 0.0,e2 0.0,e3 0.0,e4 0.0,e5 0.0,e6 0.0}
DECL FDAT FPS_36={TOOL_NO 3,BASE_NO 3,IPO_FRAME #BASE}
DECL PDAT PPDAT30={VEL 100.0,ACC 80.0,APO_DIST 100.0}
DECL E6POS XPS_37={x 190.027893,y 229.223999,z 5.26974916,a 81.5058365,b -2.0061059,c -93.3127136,s 2,t 43,e1 0.0,e2 0.0,e3 0.0,e4 0.0,e5 0.0,e6 0.0}
DECL FDAT FPS_37={TOOL_NO 3,BASE_NO 3,IPO_FRAME #BASE}
DECL PDAT PPDAT31={VEL 100.0,ACC 80.0,APO_DIST 100.0}
DECL E6POS XPS_38={x 224.422607,y 239.474503,z -38.9988289,a 81.3575516,b 2.56497407,c -89.2551422,s 2,t 43,e1 0.0,e2 0.0,e3 0.0,e4 0.0,e5 0.0,e6 0.0}
DECL FDAT FPS_38={TOOL_NO 3,BASE_NO 3,IPO_FRAME #BASE}
DECL PDAT PPDAT32={VEL 100.0,ACC 80.0,APO_DIST 100.0}
DECL E6POS XSWP_60_7106={x 183.081604,y 238.061493,z -37.7795715,a 87.6000137,b 2.26684809,c -93.2115173,s 2,t 43,e1 0.0,e2 0.0,e3 0.0,e4 0.0,e5 0.0,e6 0.0}
DECL FDAT FSWP_60_7106={TOOL_NO 3,BASE_NO 3,IPO_FRAME #BASE}
DECL LDAT LCPDAT22={VEL 2.0,ACC 100.0,APO_DIST 100.0,APO_FAC 50.0}
DECL E6POS XSWP_60_7108={x 183.750793,y 265.563995,z -27.4932194,a 87.6010666,b 2.26722002,c -93.2134781,s 2,t 43,e1 0.0,e2 0.0,e3 0.0,e4 0.0,e5 0.0,e6 0.0}
DECL FDAT FSWP_60_7108={TOOL_NO 3,BASE_NO 3,IPO_FRAME #BASE}
DECL LDAT LCPDAT23={VEL 2.0,ACC 100.0,APO_DIST 100.0,APO_FAC 50.0}
DECL E6POS XSWP_60_7110={x 184.475403,y 297.221313,z -15.1434097,a 87.5958328,b 2.26497602,c -93.2134705,s 2,t 43,e1 0.0,e2 0.0,e3 0.0,e4 0.0,e5 0.0,e6 0.0}
DECL FDAT FSWP_60_7110={TOOL_NO 3,BASE_NO 3,IPO_FRAME #BASE}
DECL LDAT LCPDAT24={VEL 2.0,ACC 100.0,APO_DIST 100.0,APO_FAC 50.0}
DECL E6POS XSWP_60_7112={x 182.128601,y 359.83139,z -0.941925526,a 87.5949631,b 2.26507401,c -93.213501,s 2,t 43,e1 0.0,e2 0.0,e3 0.0,e4 0.0,e5 0.0,e6 0.0}
DECL FDAT FSWP_60_7112={TOOL_NO 3,BASE_NO 3,IPO_FRAME #BASE}
DECL LDAT LCPDAT25={VEL 2.0,ACC 100.0,APO_DIST 100.0,APO_FAC 50.0}
DECL E6POS XSWP_60_7114={x 186.180206,y 379.217102,z 1.77508795,a 87.5944595,b 2.26477695,c -93.2110138,s 2,t 43,e1 0.0,e2 0.0,e3 0.0,e4 0.0,e5 0.0,e6 0.0}
DECL FDAT FSWP_60_7114={TOOL_NO 3,BASE_NO 3,IPO_FRAME #BASE}
DECL LDAT LCPDAT26={VEL 2.0,ACC 100.0,APO_DIST 100.0,APO_FAC 50.0}
DECL E6POS XSWP_60_7028={x 185.937897,y 359.871887,z -0.961844385,a 87.5954437,b 2.26407409,c -93.2123184,s 2,t 43,e1 0.0,e2 0.0,e3 0.0,e4 0.0,e5 0.0,e6 0.0}
DECL FDAT FSWP_60_7028={TOOL_NO 3,BASE_NO 3,IPO_FRAME #BASE}
DECL E6POS XSWP_60_7116={x 185.287094,y 414.170685,z 26.6693096,a 87.7702866,b -0.879706621,c -93.2080078,s 2,t 43,e1 0.0,e2 0.0,e3 0.0,e4 0.0,e5 0.0,e6 0.0}
DECL FDAT FSWP_60_7116={TOOL_NO 3,BASE_NO 3,IPO_FRAME #BASE}
DECL LDAT LCPDAT27={VEL 2.0,ACC 100.0,APO_DIST 100.0,APO_FAC 50.0}
DECL E6POS XSWP_60_7118={x 181.490906,y 418.84259,z 53.1533203,a 87.8234634,b -5.40211916,c -93.2266388,s 2,t 43,e1 0.0,e2 0.0,e3 0.0,e4 0.0,e5 0.0,e6 0.0}
DECL FDAT FSWP_60_7118={TOOL_NO 3,BASE_NO 3,IPO_FRAME #BASE}
DECL LDAT LCPDAT28={VEL 2.0,ACC 100.0,APO_DIST 100.0,APO_FAC 50.0}
DECL E6POS XSWP_60_7120={x 185.961304,y 420.436005,z 81.3283768,a 87.8185883,b -5.39959097,c -93.2263489,s 2,t 43,e1 0.0,e2 0.0,e3 0.0,e4 0.0,e5 0.0,e6 0.0}
DECL FDAT FSWP_60_7120={TOOL_NO 3,BASE_NO 3,IPO_FRAME #BASE}
DECL LDAT LCPDAT29={VEL 2.0,ACC 100.0,APO_DIST 100.0,APO_FAC 50.0}
DECL E6POS XSWP_60_7121={x 181.620407,y 347.470306,z 83.9234619,a 87.8192062,b -5.4038291,c -93.2219467,s 2,t 43,e1 0.0,e2 0.0,e3 0.0,e4 0.0,e5 0.0,e6 0.0}
DECL FDAT FSWP_60_7121={TOOL_NO 3,BASE_NO 3,IPO_FRAME #BASE}
DECL PDAT PPDAT33={VEL 100.0,ACC 80.0,APO_DIST 100.0}
DECL E6POS XSWP_60_7122={x 181.620407,y 347.470306,z 83.9234619,a 87.8192062,b -5.4038291,c -93.2219467,s 2,t 43,e1 0.0,e2 0.0,e3 0.0,e4 0.0,e5 0.0,e6 0.0}
DECL FDAT FSWP_60_7122={TOOL_NO 3,BASE_NO 3,IPO_FRAME #BASE}
DECL PDAT PPDAT34={VEL 100.0,ACC 80.0,APO_DIST 100.0}
DECL E6POS XSWP_60_7123={x -147.606903,y 344.160706,z 83.5968781,a 87.8187332,b -5.40472984,c -93.2222366,s 2,t 42,e1 0.0,e2 0.0,e3 0.0,e4 0.0,e5 0.0,e6 0.0}
DECL FDAT FSWP_60_7123={TOOL_NO 3,BASE_NO 3,IPO_FRAME #BASE}
DECL PDAT PPDAT35={VEL 100.0,ACC 80.0,APO_DIST 100.0}
DECL E6POS XSWP_60_7124={x -373.179199,y 990.898926,z -71.8238373,a 96.4663162,b 6.40630579,c -88.1937637,s 2,t 42,e1 0.0,e2 0.0,e3 0.0,e4 0.0,e5 0.0,e6 0.0}
DECL FDAT FSWP_60_7124={TOOL_NO 3,BASE_NO 3,IPO_FRAME #BASE}
DECL PDAT PPDAT36={VEL 100.0,ACC 80.0,APO_DIST 100.0}
DECL E6POS XSWP_60_7125={x -938.606628,y 703.750183,z 612.628296,a 165.017105,b 23.1202908,c 13.1029396,s 2,t 42,e1 0.0,e2 0.0,e3 0.0,e4 0.0,e5 0.0,e6 0.0}
DECL FDAT FSWP_60_7125={TOOL_NO 3,BASE_NO 3,IPO_FRAME #BASE}
DECL PDAT PPDAT37={VEL 100.0,ACC 80.0,APO_DIST 100.0}
DECL E6POS XSWP_60_7126={x -936.03772,y 1095.39502,z 612.167786,a 165.015793,b 23.1197605,c 13.09867,s 2,t 43,e1 0.0,e2 0.0,e3 0.0,e4 0.0,e5 0.0,e6 0.0}
DECL FDAT FSWP_60_7126={TOOL_NO 3,BASE_NO 3,IPO_FRAME #BASE}
DECL PDAT PPDAT38={VEL 100.0,ACC 80.0,APO_DIST 100.0}
DECL E6POS XSWP_60_7234={x 205.6577,y 368.187012,z 389.243713,a -89.9944229,b 62.69561,c 90.0030975,s 2,t 43,e1 0.0,e2 0.0,e3 0.0,e4 0.0,e5 0.0,e6 0.0}
DECL FDAT FSWP_60_7234={TOOL_NO 3,BASE_NO 3,IPO_FRAME #BASE}
DECL E6POS XSWP_60_7228={x 206.997299,y 237.645493,z 384.287994,a -90.0011597,b 62.6945915,c 89.9988098,s 2,t 43,e1 0.0,e2 0.0,e3 0.0,e4 0.0,e5 0.0,e6 0.0}
DECL FDAT FSWP_60_7228={TOOL_NO 3,BASE_NO 3,IPO_FRAME #BASE}
DECL E6POS XSWP_60_7226={x 207.525299,y 187.710403,z 383.361206,a -90.0016327,b 62.6922607,c 89.9979324,s 2,t 43,e1 0.0,e2 0.0,e3 0.0,e4 0.0,e5 0.0,e6 0.0}
DECL FDAT FSWP_60_7226={TOOL_NO 3,BASE_NO 3,IPO_FRAME #BASE}
DECL E6POS XSWP_60_7224={x 206.951508,y 141.325897,z 384.747589,a -89.9992218,b 54.2501106,c 89.9959335,s 2,t 43,e1 0.0,e2 0.0,e3 0.0,e4 0.0,e5 0.0,e6 0.0}
DECL FDAT FSWP_60_7224={TOOL_NO 3,BASE_NO 3,IPO_FRAME #BASE}
DECL E6POS XSWP_60_7250={x 180.742096,y 249.745895,z 487.002686,a -73.5239868,b 45.4169807,c 112.489998,s 2,t 11,e1 0.0,e2 0.0,e3 0.0,e4 0.0,e5 0.0,e6 0.0}
DECL FDAT FSWP_60_7250={TOOL_NO 3,BASE_NO 3,IPO_FRAME #BASE}
DECL E6POS XSWP_60_9324={x 211.497406,y 837.818176,z 419.146515,a -89.9909286,b 86.8919983,c 90.0067215,s 2,t 43,e1 0.0,e2 0.0,e3 0.0,e4 0.0,e5 0.0,e6 0.0}
DECL FDAT FSWP_60_9324={TOOL_NO 3,BASE_NO 3,IPO_FRAME #BASE}
DECL E6POS XSWP_60_9326={x 209.523499,y 813.088623,z 427.234314,a -90.0934982,b 86.8950806,c 89.9074478,s 2,t 43,e1 0.0,e2 0.0,e3 0.0,e4 0.0,e5 0.0,e6 0.0}
DECL FDAT FSWP_60_9326={TOOL_NO 3,BASE_NO 3,IPO_FRAME #BASE}
DECL E6POS XSWP_60_9328={x 210.7603,y 785.246887,z 444.832489,a -90.0749817,b 86.8963165,c 89.9261932,s 2,t 43,e1 0.0,e2 0.0,e3 0.0,e4 0.0,e5 0.0,e6 0.0}
DECL FDAT FSWP_60_9328={TOOL_NO 3,BASE_NO 3,IPO_FRAME #BASE}
DECL E6POS XSWP_60_9330={x 213.020096,y 756.550476,z 466.476013,a -90.016777,b 86.8942871,c 89.982933,s 2,t 43,e1 0.0,e2 0.0,e3 0.0,e4 0.0,e5 0.0,e6 0.0}
DECL FDAT FSWP_60_9330={TOOL_NO 3,BASE_NO 3,IPO_FRAME #BASE}
DECL E6POS XSWP_60_9332={x 211.718094,y 725.370728,z 475.666199,a 90.0008621,b 70.9207306,c -89.9995728,s 2,t 43,e1 0.0,e2 0.0,e3 0.0,e4 0.0,e5 0.0,e6 0.0}
DECL FDAT FSWP_60_9332={TOOL_NO 3,BASE_NO 3,IPO_FRAME #BASE}
DECL E6POS XSWP_60_9334={x 210.650497,y 692.968994,z 480.713409,a -90.0100098,b 86.1567688,c 89.9899673,s 2,t 43,e1 0.0,e2 0.0,e3 0.0,e4 0.0,e5 0.0,e6 0.0}
DECL FDAT FSWP_60_9334={TOOL_NO 3,BASE_NO 3,IPO_FRAME #BASE}
DECL E6POS XSWP_60_9336={x 211.194305,y 660.460876,z 480.689911,a -89.9966736,b 56.1083107,c 90.0018005,s 2,t 43,e1 0.0,e2 0.0,e3 0.0,e4 0.0,e5 0.0,e6 0.0}
DECL FDAT FSWP_60_9336={TOOL_NO 3,BASE_NO 3,IPO_FRAME #BASE}
DECL E6POS XSWP_60_9338={x 210.866592,y 634.383301,z 481.291992,a -90.0009232,b 58.2448807,c 90.0010529,s 2,t 43,e1 0.0,e2 0.0,e3 0.0,e4 0.0,e5 0.0,e6 0.0}
DECL FDAT FSWP_60_9338={TOOL_NO 3,BASE_NO 3,IPO_FRAME #BASE}
DECL E6POS XSWP_60_9340={x 210.658401,y 608.414612,z 481.042114,a -90.0021362,b 59.0431213,c 89.9979324,s 2,t 43,e1 0.0,e2 0.0,e3 0.0,e4 0.0,e5 0.0,e6 0.0}
DECL FDAT FSWP_60_9340={TOOL_NO 3,BASE_NO 3,IPO_FRAME #BASE}
DECL E6POS XSWP_60_9342={x 211.162201,y 582.413513,z 480.874298,a -90.0032883,b 59.72015,c 89.9965363,s 2,t 43,e1 0.0,e2 0.0,e3 0.0,e4 0.0,e5 0.0,e6 0.0}
DECL FDAT FSWP_60_9342={TOOL_NO 3,BASE_NO 3,IPO_FRAME #BASE}
DECL E6POS XSWP_60_9344={x 211.489395,y 556.442871,z 480.0336,a -90.0012436,b 60.0731697,c 89.9978027,s 2,t 43,e1 0.0,e2 0.0,e3 0.0,e4 0.0,e5 0.0,e6 0.0}
DECL FDAT FSWP_60_9344={TOOL_NO 3,BASE_NO 3,IPO_FRAME #BASE}
DECL E6POS XSWP_60_9214={x 209.414597,y 441.113495,z 482.718414,a -89.9964828,b 60.0045891,c 90.000679,s 2,t 43,e1 0.0,e2 0.0,e3 0.0,e4 0.0,e5 0.0,e6 0.0}
DECL FDAT FSWP_60_9214={TOOL_NO 3,BASE_NO 3,IPO_FRAME #BASE}
DECL E6POS XSWP_60_9210={x 211.829102,y 431.055115,z 441.071014,a -89.9971771,b 61.5311394,c 90.0033798,s 2,t 43,e1 0.0,e2 0.0,e3 0.0,e4 0.0,e5 0.0,e6 0.0}
DECL FDAT FSWP_60_9210={TOOL_NO 3,BASE_NO 3,IPO_FRAME #BASE}
DECL E6POS XSWP_60_9208={x 212.199097,y 416.683685,z 400.172302,a -90.0129471,b 62.6884308,c 89.9872208,s 2,t 43,e1 0.0,e2 0.0,e3 0.0,e4 0.0,e5 0.0,e6 0.0}
DECL FDAT FSWP_60_9208={TOOL_NO 3,BASE_NO 3,IPO_FRAME #BASE}
DECL E6POS XSWP_60_9218={x 212.7341,y 88.1504822,z 383.971893,a -89.998497,b 44.4745903,c 89.9906387,s 2,t 43,e1 0.0,e2 0.0,e3 0.0,e4 0.0,e5 0.0,e6 0.0}
DECL FDAT FSWP_60_9218={TOOL_NO 3,BASE_NO 3,IPO_FRAME #BASE}
DECL E6POS XSWP_60_9216={x 212.939194,y 39.3732491,z 383.035004,a -89.9955826,b 44.4738083,c 89.9938278,s 2,t 43,e1 0.0,e2 0.0,e3 0.0,e4 0.0,e5 0.0,e6 0.0}
DECL FDAT FSWP_60_9216={TOOL_NO 3,BASE_NO 3,IPO_FRAME #BASE}
DECL E6POS XSWP_60_9257={x 186.411804,y -3.74332094,z 490.071991,a -80.9862213,b 30.2953091,c 107.447701,s 2,t 11,e1 0.0,e2 0.0,e3 0.0,e4 0.0,e5 0.0,e6 0.0}
DECL FDAT FSWP_60_9257={TOOL_NO 3,BASE_NO 3,IPO_FRAME #BASE}
DECL E6POS XSWP_60_9256={x 184.425003,y 50.293541,z 489.944489,a -80.3128433,b 32.1282997,c 107.793503,s 2,t 11,e1 0.0,e2 0.0,e3 0.0,e4 0.0,e5 0.0,e6 0.0}
DECL FDAT FSWP_60_9256={TOOL_NO 3,BASE_NO 3,IPO_FRAME #BASE}
DECL E6POS XSWP_60_9254={x 185.411102,y 92.7307968,z 490.32019,a -80.3133774,b 32.1280289,c 107.791603,s 2,t 11,e1 0.0,e2 0.0,e3 0.0,e4 0.0,e5 0.0,e6 0.0}
DECL FDAT FSWP_60_9254={TOOL_NO 3,BASE_NO 3,IPO_FRAME #BASE}
DECL E6POS XSWP_60_9234={x 204.064499,y 385.707397,z 414.247314,a -43.1890182,b 69.0715637,c 138.712708,s 2,t 43,e1 0.0,e2 0.0,e3 0.0,e4 0.0,e5 0.0,e6 0.0}
DECL FDAT FSWP_60_9234={TOOL_NO 3,BASE_NO 3,IPO_FRAME #BASE}
DECL LDAT LCPDAT30={VEL 2.0,ACC 100.0,APO_DIST 100.0,APO_FAC 50.0}
ENDDAT
